LIN {X 0,Y 489.768,Z 496.866,A -85,B 0,C 180,E1 -6554.925,E2 -6554.925} C_VEL
LIN {X 0,Y 489.271,Z 508.598,A -85,B 0,C 180,E1 -6556.29,E2 -6556.29} C_VEL
LIN {X 0,Y 488.822,Z 518.89,A -85,B 0,C 180,E1 -6557.728,E2 -6557.728} C_VEL
LIN {X 0,Y 488.607,Z 527.81,A -85,B 0,C 180,E1 -6559.223,E2 -6559.223} C_VEL
LIN {X 0,Y 488.258,Z 535.963,A -85,B 0,C 180,E1 -6560.89,E2 -6560.89} C_VEL
LIN {X 0,Y 488.146,Z 542.468,A -85,B 0,C 180,E1 -6562.555,E2 -6562.555} C_VEL
LIN {X 0,Y 488.093,Z 547.498,A -85,B 0,C 180,E1 -6564.215,E2 -6564.215} C_VEL
LIN {X 0,Y 488.046,Z 551.175,A -85,B 0,C 180,E1 -6565.871,E2 -6565.871} C_VEL
LIN {X 0,Y 488.011,Z 553.582,A -85,B 0,C 180,E1 -6567.524,E2 -6567.524} C_VEL
LIN {X 0,Y 487.933,Z 554.765,A -85,B 0,C 180,E1 -6569.175,E2 -6569.175} C_VEL
LIN {X 0,Y 487.937,Z 554.732,A -85,B 0,C 180,E1 -6570.825,E2 -6570.825} C_VEL
LIN {X 0,Y 488.021,Z 553.482,A -85,B 0,C 180,E1 -6572.476,E2 -6572.476} C_VEL
LIN {X 0,Y 488.083,Z 551.011,A -85,B 0,C 180,E1 -6574.129,E2 -6574.129} C_VEL
LIN {X 0,Y 488.118,Z 547.258,A -85,B 0,C 180,E1 -6575.785,E2 -6575.785} C_VEL
LIN {X 0,Y 488.183,Z 542.13,A -85,B 0,C 180,E1 -6577.445,E2 -6577.445} C_VEL
LIN {X 0,Y 488.289,Z 535.484,A -85,B 0,C 180,E1 -6579.11,E2 -6579.11} C_VEL
LIN {X 0,Y 488.567,Z 528.339,A -85,B 0,C 180,E1 -6580.569,E2 -6580.569} C_VEL
LIN {X 0,Y 488.758,Z 519.247,A -85,B 0,C 180,E1 -6582.098,E2 -6582.098} C_VEL
LIN {X 0,Y 489.278,Z 507.782,A -85,B 0,C 180,E1 -6583.71,E2 -6583.71} C_VEL
LIN {X 0,Y 489.719,Z 497.109,A -85,B 0,C 180,E1 -6584.971,E2 -6584.971} C_VEL
LIN {X 0,Y 490.258,Z 486.421,A -85,B 0,C 180,E1 -6586.042,E2 -6586.042} C_VEL
LIN {X 0,Y 490.91,Z 472.849,A -85,B 0,C 180,E1 -6587.174,E2 -6587.174} C_VEL
LIN {X 0,Y 491.491,Z 460.708,A -85,B 0,C 180,E1 -6588.013,E2 -6588.013} C_VEL
LIN {X 0,Y 492.097,Z 446.698,A -85,B 0,C 180,E1 -6588.798,E2 -6588.798} C_VEL
LIN {X 0,Y 492.623,Z 432.142,A -85,B 0,C 180,E1 -6589.434,E2 -6589.434} C_VEL
LIN {X 0,Y 493.083,Z 417.146,A -85,B 0,C 180,E1 -6589.914,E2 -6589.914} C_VEL
LIN {X 0,Y 492.97,Z 413.138,A -85,B 0,C 180,E1 -6590.021,E2 -6590.021} C_VEL
LIN {X 0,Y 491.062,Z 401.561,A -85,B 0,C 180,E1 -6590.337,E2 -6590.337} C_VEL
LIN {X 0,Y 489.673,Z 391.28,A -85,B 0,C 180,E1 -6590.556,E2 -6590.556} C_VEL
LIN {X 0,Y 490.143,Z 374.363,A -85,B 0,C 180,E1 -6593.412,E2 -6593.412} C_VEL
LIN {X 0,Y 490.901,Z 356.546,A -85,B 0,C 180,E1 -6596.577,E2 -6596.577} C_VEL
LIN {X 0,Y 491.916,Z 340.726,A -85,B 0,C 180,E1 -6599.609,E2 -6599.609} C_VEL
LIN {X 0,Y 493.222,Z 326.855,A -85,B 0,C 180,E1 -6602.541,E2 -6602.541} C_VEL
LIN {X 0,Y 494.841,Z 316.102,A -85,B 0,C 180,E1 -6605.114,E2 -6605.114} C_VEL
LIN {X 0,Y 494.625,Z 313.33,A -85,B 0,C 180,E1 -6605.914,E2 -6605.914} C_VEL
LIN {X 0,Y 493.242,Z 307.964,A -85,B 0,C 180,E1 -6607.784,E2 -6607.784} C_VEL
LIN {X 0,Y 491.895,Z 302.8,A -85,B 0,C 180,E1 -6610.012,E2 -6610.012} C_VEL
LIN {X 0,Y 490.897,Z 299.006,A -85,B 0,C 180,E1 -6612.29,E2 -6612.29} C_VEL
LIN {X 0,Y 490.311,Z 296.887,A -85,B 0,C 180,E1 -6614.218,E2 -6614.218} C_VEL
LIN {X 0,Y 489.902,Z 295.578,A -85,B 0,C 180,E1 -6616.481,E2 -6616.481} C_VEL
LIN {X 0,Y 489.802,Z 295.249,A -85,B 0,C 180,E1 -6618.697,E2 -6618.697} C_VEL
LIN {X 0,Y 489.783,Z 295.681,A -85,B 0,C 180,E1 -6620.849,E2 -6620.849} C_VEL
LIN {X 0,Y 489.826,Z 296.807,A -85,B 0,C 180,E1 -6623.465,E2 -6623.465} C_VEL
LIN {X 0,Y 489.686,Z 298.58,A -85,B 0,C 180,E1 -6626.349,E2 -6626.349} C_VEL
LIN {X 0,Y 489.42,Z 300.813,A -85,B 0,C 180,E1 -6629.496,E2 -6629.496} C_VEL
LIN {X 0,Y 489.329,Z 302.428,A -85,B 0,C 180,E1 -6631.708,E2 -6631.708} C_VEL
LIN {X 0,Y 489.182,Z 304.804,A -85,B 0,C 180,E1 -6634.839,E2 -6634.839} C_VEL
LIN {X 0,Y 489.027,Z 307.367,A -85,B 0,C 180,E1 -6638.059,E2 -6638.059} C_VEL
LIN {X 0,Y 488.915,Z 309.511,A -85,B 0,C 180,E1 -6640.694,E2 -6640.694} C_VEL
LIN {X 0,Y 488.801,Z 311.695,A -85,B 0,C 180,E1 -6643.288,E2 -6643.288} C_VEL
LIN {X 0,Y 488.772,Z 313.227,A -85,B 0,C 180,E1 -6645.04,E2 -6645.04} C_VEL
LIN {X 0,Y 492.021,Z 323.275,A -85,B 0,C 180,E1 -6645.508,E2 -6645.508} C_VEL
LIN {X 0,Y 491.727,Z 335.772,A -85,B 0,C 180,E1 -6646.044,E2 -6646.044} C_VEL
LIN {X 0,Y 491.293,Z 348.473,A -85,B 0,C 180,E1 -6646.769,E2 -6646.769} C_VEL
LIN {X 0,Y 490.795,Z 359.859,A -85,B 0,C 180,E1 -6647.597,E2 -6647.597} C_VEL
LIN {X 0,Y 490.344,Z 371.117,A -85,B 0,C 180,E1 -6648.634,E2 -6648.634} C_VEL
LIN {X 0,Y 489.981,Z 380.286,A -85,B 0,C 180,E1 -6649.672,E2 -6649.672} C_VEL
LIN {X 0,Y 489.607,Z 387.86,A -85,B 0,C 180,E1 -6650.707,E2 -6650.707} C_VEL
LIN {X 0,Y 489.263,Z 395.396,A -85,B 0,C 180,E1 -6651.97,E2 -6651.97} C_VEL
LIN {X 0,Y 489.024,Z 402.088,A -85,B 0,C 180,E1 -6653.398,E2 -6653.398} C_VEL
LIN {X 0,Y 488.756,Z 406.626,A -85,B 0,C 180,E1 -6654.637,E2 -6654.637} C_VEL
LIN {X 0,Y 488.595,Z 410.068,A -85,B 0,C 180,E1 -6655.876,E2 -6655.876} C_VEL
LIN {X 0,Y 488.644,Z 411.805,A -85,B 0,C 180,E1 -6656.702,E2 -6656.702} C_VEL
LIN {X 0,Y 488.49,Z 413.141,A -85,B 0,C 180,E1 -6657.526,E2 -6657.526} C_VEL
LIN {X 0,Y 488.382,Z 414.052,A -85,B 0,C 180,E1 -6658.351,E2 -6658.351} C_VEL
LIN {X 0,Y 488.402,Z 414.706,A -85,B 0,C 180,E1 -6660,E2 -6660} C_VEL
LIN {X 0,Y 488.403,Z 414.441,A -85,B 0,C 180,E1 -6660.825,E2 -6660.825} C_VEL
LIN {X 0,Y 488.32,Z 412.723,A -85,B 0,C 180,E1 -6662.475,E2 -6662.475} C_VEL
LIN {X 0,Y 488.395,Z 411.27,A -85,B 0,C 180,E1 -6663.3,E2 -6663.3} C_VEL
LIN {X 0,Y 488.539,Z 408.258,A -85,B 0,C 180,E1 -6664.538,E2 -6664.538} C_VEL
LIN {X 0,Y 488.575,Z 404.251,A -85,B 0,C 180,E1 -6665.779,E2 -6665.779} C_VEL
LIN {X 0,Y 488.792,Z 399.728,A -85,B 0,C 180,E1 -6666.879,E2 -6666.879} C_VEL
LIN {X 0,Y 489.007,Z 392.666,A -85,B 0,C 180,E1 -6668.263,E2 -6668.263} C_VEL
LIN {X 0,Y 489.314,Z 384.64,A -85,B 0,C 180,E1 -6669.507,E2 -6669.507} C_VEL
LIN {X 0,Y 489.599,Z 376.5,A -85,B 0,C 180,E1 -6670.546,E2 -6670.546} C_VEL
LIN {X 0,Y 490.05,Z 366.603,A -85,B 0,C 180,E1 -6671.583,E2 -6671.583} C_VEL
LIN {X 0,Y 490.437,Z 355.629,A -85,B 0,C 180,E1 -6672.518,E2 -6672.518} C_VEL
LIN {X 0,Y 490.801,Z 343.259,A -85,B 0,C 180,E1 -6673.35,E2 -6673.35} C_VEL
LIN {X 0,Y 491.123,Z 331.319,A -85,B 0,C 180,E1 -6673.974,E2 -6673.974} C_VEL
LIN {X 0,Y 491.176,Z 320.509,A -85,B 0,C 180,E1 -6674.409,E2 -6674.409} C_VEL
LIN {X 0,Y 488.179,Z 308.882,A -85,B 0,C 180,E1 -6674.859,E2 -6674.859} C_VEL
LIN {X 0,Y 488.179,Z 305.272,A -85,B 0,C 180,E1 -6678.165,E2 -6678.165} C_VEL
LIN {X 0,Y 488.206,Z 302.102,A -85,B 0,C 180,E1 -6681.093,E2 -6681.093} C_VEL
LIN {X 0,Y 488.197,Z 299.235,A -85,B 0,C 180,E1 -6683.771,E2 -6683.771} C_VEL
LIN {X 0,Y 488.232,Z 296.325,A -85,B 0,C 180,E1 -6686.503,E2 -6686.503} C_VEL
LIN {X 0,Y 488.278,Z 293.326,A -85,B 0,C 180,E1 -6689.3,E2 -6689.3} C_VEL
LIN {X 0,Y 488.267,Z 290.293,A -85,B 0,C 180,E1 -6692.179,E2 -6692.179} C_VEL
LIN {X 0,Y 488.605,Z 290.25,A -85,B 0,C 180,E1 -6695.124,E2 -6695.124} C_VEL
LIN {X 0,Y 488.681,Z 290.235,A -85,B 0,C 180,E1 -6698.2,E2 -6698.2} C_VEL
LIN {X 0,Y 488.721,Z 290.231,A -85,B 0,C 180,E1 -6700.345,E2 -6700.345} C_VEL
LIN {X 0,Y 488.687,Z 290.233,A -85,B 0,C 180,E1 -6703.655,E2 -6703.655} C_VEL
LIN {X 0,Y 488.676,Z 290.241,A -85,B 0,C 180,E1 -6706.344,E2 -6706.344} C_VEL
LIN {X 0,Y 488.631,Z 290.247,A -85,B 0,C 180,E1 -6708.576,E2 -6708.576} C_VEL
LIN {X 0,Y 488.638,Z 290.577,A -85,B 0,C 180,E1 -6709.667,E2 -6709.667} C_VEL
LIN {X 0,Y 488.639,Z 294.469,A -85,B 0,C 180,E1 -6712.284,E2 -6712.284} C_VEL
LIN {X 0,Y 488.59,Z 298.405,A -85,B 0,C 180,E1 -6715.075,E2 -6715.075} C_VEL
LIN {X 0,Y 488.542,Z 302.488,A -85,B 0,C 180,E1 -6718.077,E2 -6718.077} C_VEL
LIN {X 0,Y 488.447,Z 305.354,A -85,B 0,C 180,E1 -6720.198,E2 -6720.198} C_VEL
LIN {X 0,Y 487.763,Z 306.347,A -85,B 0,C 180,E1 -6720.877,E2 -6720.877} C_VEL
LIN {X 0,Y 484.894,Z 308.223,A -85,B 0,C 180,E1 -6721.972,E2 -6721.972} C_VEL
LIN {X 0,Y 482.476,Z 309.764,A -85,B 0,C 180,E1 -6722.855,E2 -6722.855} C_VEL
LIN {X 0,Y 481.436,Z 310.86,A -85,B 0,C 180,E1 -6723.538,E2 -6723.538} C_VEL
LIN {X 0,Y 481.351,Z 311.192,A -85,B 0,C 180,E1 -6723.77,E2 -6723.77} C_VEL
LIN {X 0,Y 481.32,Z 315.603,A -85,B 0,C 180,E1 -6726.781,E2 -6726.781} C_VEL
LIN {X 0,Y 481.337,Z 318.973,A -85,B 0,C 180,E1 -6728.946,E2 -6728.946} C_VEL
LIN {X 0,Y 486.935,Z 336.217,A -85,B 0,C 180,E1 -6729.595,E2 -6729.595} C_VEL
LIN {X 0,Y 487.422,Z 339.11,A -85,B 0,C 180,E1 -6729.704,E2 -6729.704} C_VEL
LIN {X 0,Y 487.036,Z 354.063,A -85,B 0,C 180,E1 -6730.234,E2 -6730.234} C_VEL
LIN {X 0,Y 486.428,Z 368.55,A -85,B 0,C 180,E1 -6730.92,E2 -6730.92} C_VEL
LIN {X 0,Y 485.761,Z 382.515,A -85,B 0,C 180,E1 -6731.767,E2 -6731.767} C_VEL
LIN {X 0,Y 485.028,Z 395.249,A -85,B 0,C 180,E1 -6732.72,E2 -6732.72} C_VEL
LIN {X 0,Y 484.313,Z 407.382,A -85,B 0,C 180,E1 -6733.82,E2 -6733.82} C_VEL
LIN {X 0,Y 483.565,Z 418.712,A -85,B 0,C 180,E1 -6735.05,E2 -6735.05} C_VEL
LIN {X 0,Y 482.977,Z 428.555,A -85,B 0,C 180,E1 -6736.322,E2 -6736.322} C_VEL
LIN {X 0,Y 482.399,Z 437.227,A -85,B 0,C 180,E1 -6737.651,E2 -6737.651} C_VEL
LIN {X 0,Y 481.895,Z 446.114,A -85,B 0,C 180,E1 -6739.283,E2 -6739.283} C_VEL
LIN {X 0,Y 481.547,Z 452.691,A -85,B 0,C 180,E1 -6740.761,E2 -6740.761} C_VEL
LIN {X 0,Y 481.289,Z 458.773,A -85,B 0,C 180,E1 -6742.448,E2 -6742.448} C_VEL
LIN {X 0,Y 481.097,Z 463.478,A -85,B 0,C 180,E1 -6744.131,E2 -6744.131} C_VEL
LIN {X 0,Y 480.997,Z 466.926,A -85,B 0,C 180,E1 -6745.81,E2 -6745.81} C_VEL
LIN {X 0,Y 480.935,Z 469.203,A -85,B 0,C 180,E1 -6747.487,E2 -6747.487} C_VEL
LIN {X 0,Y 480.799,Z 470.371,A -85,B 0,C 180,E1 -6749.162,E2 -6749.162} C_VEL
LIN {X 0,Y 480.798,Z 470.387,A -85,B 0,C 180,E1 -6750.837,E2 -6750.837} C_VEL
LIN {X 0,Y 480.935,Z 469.281,A -85,B 0,C 180,E1 -6752.512,E2 -6752.512} C_VEL
LIN {X 0,Y 480.997,Z 467.072,A -85,B 0,C 180,E1 -6754.189,E2 -6754.189} C_VEL
LIN {X 0,Y 481.093,Z 463.7,A -85,B 0,C 180,E1 -6755.869,E2 -6755.869} C_VEL
LIN {X 0,Y 481.287,Z 459.071,A -85,B 0,C 180,E1 -6757.552,E2 -6757.552} C_VEL
LIN {X 0,Y 481.526,Z 453.061,A -85,B 0,C 180,E1 -6759.239,E2 -6759.239} C_VEL
LIN {X 0,Y 481.936,Z 445.488,A -85,B 0,C 180,E1 -6760.928,E2 -6760.928} C_VEL
LIN {X 0,Y 482.375,Z 437.935,A -85,B 0,C 180,E1 -6762.323,E2 -6762.323} C_VEL
LIN {X 0,Y 482.932,Z 429.171,A -85,B 0,C 180,E1 -6763.679,E2 -6763.679} C_VEL
LIN {X 0,Y 483.552,Z 419.434,A -85,B 0,C 180,E1 -6764.95,E2 -6764.95} C_VEL
LIN {X 0,Y 484.243,Z 408.371,A -85,B 0,C 180,E1 -6766.17,E2 -6766.17} C_VEL
LIN {X 0,Y 485.004,Z 396.286,A -85,B 0,C 180,E1 -6767.281,E2 -6767.281} C_VEL
LIN {X 0,Y 485.703,Z 383.774,A -85,B 0,C 180,E1 -6768.234,E2 -6768.234} C_VEL
LIN {X 0,Y 486.312,Z 370.13,A -85,B 0,C 180,E1 -6769.085,E2 -6769.085} C_VEL
LIN {X 0,Y 486.971,Z 355.986,A -85,B 0,C 180,E1 -6769.774,E2 -6769.774} C_VEL
LIN {X 0,Y 487.378,Z 341.683,A -85,B 0,C 180,E1 -6770.306,E2 -6770.306} C_VEL
LIN {X 0,Y 487.231,Z 337.436,A -85,B 0,C 180,E1 -6770.449,E2 -6770.449} C_VEL
LIN {X 0,Y 483.022,Z 324.071,A -85,B 0,C 180,E1 -6770.962,E2 -6770.962} C_VEL
LIN {X 0,Y 481.339,Z 318.996,A -85,B 0,C 180,E1 -6771.14,E2 -6771.14} C_VEL
LIN {X 0,Y 481.312,Z 314.379,A -85,B 0,C 180,E1 -6774.132,E2 -6774.132} C_VEL
LIN {X 0,Y 481.401,Z 310.161,A -85,B 0,C 180,E1 -6777.058,E2 -6777.058} C_VEL
LIN {X 0,Y 481.418,Z 306.456,A -85,B 0,C 180,E1 -6779.759,E2 -6779.759} C_VEL
LIN {X 0,Y 481.49,Z 302.545,A -85,B 0,C 180,E1 -6782.688,E2 -6782.688} C_VEL
LIN {X 0,Y 481.548,Z 298.434,A -85,B 0,C 180,E1 -6785.717,E2 -6785.717} C_VEL
LIN {X 0,Y 481.643,Z 293.949,A -85,B 0,C 180,E1 -6788.862,E2 -6788.862} C_VEL
LIN {X 0,Y 481.548,Z 291.136,A -85,B 0,C 180,E1 -6790.806,E2 -6790.806} C_VEL
LIN {X 0,Y 481.622,Z 291.12,A -85,B 0,C 180,E1 -6793.302,E2 -6793.302} C_VEL
LIN {X 0,Y 481.659,Z 291.116,A -85,B 0,C 180,E1 -6795.641,E2 -6795.641} C_VEL
LIN {X 0,Y 481.657,Z 291.114,A -85,B 0,C 180,E1 -6798.958,E2 -6798.958} C_VEL
LIN {X 0,Y 481.652,Z 291.117,A -85,B 0,C 180,E1 -6801.993,E2 -6801.993} C_VEL
LIN {X 0,Y 481.691,Z 291.111,A -85,B 0,C 180,E1 -6805.318,E2 -6805.318} C_VEL
LIN {X 0,Y 481.644,Z 291.116,A -85,B 0,C 180,E1 -6808.311,E2 -6808.311} C_VEL
LIN {X 0,Y 481.657,Z 291.111,A -85,B 0,C 180,E1 -6811.216,E2 -6811.216} C_VEL
LIN {X 0,Y 481.646,Z 291.11,A -85,B 0,C 180,E1 -6814.04,E2 -6814.04} C_VEL
LIN {X 0,Y 481.675,Z 291.113,A -85,B 0,C 180,E1 -6816.812,E2 -6816.812} C_VEL
LIN {X 0,Y 481.695,Z 291.104,A -85,B 0,C 180,E1 -6819.503,E2 -6819.503} C_VEL
LIN {X 0,Y 481.682,Z 291.105,A -85,B 0,C 180,E1 -6822.157,E2 -6822.157} C_VEL
LIN {X 0,Y 481.745,Z 291.099,A -85,B 0,C 180,E1 -6824.776,E2 -6824.776} C_VEL
LIN {X 0,Y 481.752,Z 291.095,A -85,B 0,C 180,E1 -6828.215,E2 -6828.215} C_VEL
LIN {X 0,Y 481.73,Z 291.105,A -85,B 0,C 180,E1 -6831.611,E2 -6831.611} C_VEL
LIN {X 0,Y 481.786,Z 291.089,A -85,B 0,C 180,E1 -6834.139,E2 -6834.139} C_VEL
LIN {X 0,Y 481.926,Z 291.077,A -85,B 0,C 180,E1 -6837.492,E2 -6837.492} C_VEL
LIN {X 0,Y 481.942,Z 291.069,A -85,B 0,C 180,E1 -6840,E2 -6840} C_VEL
LIN {X 0,Y 481.918,Z 291.079,A -85,B 0,C 180,E1 -6842.507,E2 -6842.507} C_VEL
LIN {X 0,Y 481.785,Z 291.09,A -85,B 0,C 180,E1 -6845.861,E2 -6845.861} C_VEL
LIN {X 0,Y 481.742,Z 291.104,A -85,B 0,C 180,E1 -6848.389,E2 -6848.389} C_VEL
LIN {X 0,Y 481.751,Z 291.094,A -85,B 0,C 180,E1 -6851.785,E2 -6851.785} C_VEL
LIN {X 0,Y 481.738,Z 291.101,A -85,B 0,C 180,E1 -6855.224,E2 -6855.224} C_VEL
LIN {X 0,Y 481.709,Z 291.109,A -85,B 0,C 180,E1 -6858.722,E2 -6858.722} C_VEL
LIN {X 0,Y 481.646,Z 291.108,A -85,B 0,C 180,E1 -6861.395,E2 -6861.395} C_VEL
LIN {X 0,Y 481.648,Z 291.113,A -85,B 0,C 180,E1 -6864.115,E2 -6864.115} C_VEL
LIN {X 0,Y 481.675,Z 291.108,A -85,B 0,C 180,E1 -6867.122,E2 -6867.122} C_VEL
LIN {X 0,Y 481.673,Z 291.11,A -85,B 0,C 180,E1 -6869.741,E2 -6869.741} C_VEL
LIN {X 0,Y 481.672,Z 291.109,A -85,B 0,C 180,E1 -6872.674,E2 -6872.674} C_VEL
LIN {X 0,Y 481.66,Z 291.115,A -85,B 0,C 180,E1 -6875.204,E2 -6875.204} C_VEL
LIN {X 0,Y 481.666,Z 291.113,A -85,B 0,C 180,E1 -6878.859,E2 -6878.859} C_VEL
LIN {X 0,Y 481.652,Z 291.112,A -85,B 0,C 180,E1 -6881.913,E2 -6881.913} C_VEL
LIN {X 0,Y 481.654,Z 291.109,A -85,B 0,C 180,E1 -6884.458,E2 -6884.458} C_VEL
LIN {X 0,Y 481.628,Z 291.112,A -85,B 0,C 180,E1 -6887.837,E2 -6887.837} C_VEL
LIN {X 0,Y 481.646,Z 291.215,A -85,B 0,C 180,E1 -6888.591,E2 -6888.591} C_VEL
LIN {X 0,Y 484.909,Z 303.856,A -85,B 0,C 180,E1 -6891.801,E2 -6891.801} C_VEL
LIN {X 0,Y 487.48,Z 314.226,A -85,B 0,C 180,E1 -6894.278,E2 -6894.278} C_VEL
LIN {X 0,Y 487.662,Z 316.627,A -85,B 0,C 180,E1 -6894.798,E2 -6894.798} C_VEL
LIN {X 0,Y 486.351,Z 332.215,A -85,B 0,C 180,E1 -6897.924,E2 -6897.924} C_VEL
LIN {X 0,Y 485.178,Z 347.976,A -85,B 0,C 180,E1 -6900.971,E2 -6900.971} C_VEL
LIN {X 0,Y 484.134,Z 365.065,A -85,B 0,C 180,E1 -6904.162,E2 -6904.162} C_VEL
LIN {X 0,Y 483.249,Z 382.552,A -85,B 0,C 180,E1 -6907.332,E2 -6907.332} C_VEL
LIN {X 0,Y 482.896,Z 392.937,A -85,B 0,C 180,E1 -6909.176,E2 -6909.176} C_VEL
LIN {X 0,Y 485.472,Z 409.983,A -85,B 0,C 180,E1 -6909.592,E2 -6909.592} C_VEL
LIN {X 0,Y 486.389,Z 416.005,A -85,B 0,C 180,E1 -6909.781,E2 -6909.781} C_VEL
LIN {X 0,Y 485.948,Z 429.67,A -85,B 0,C 180,E1 -6910.213,E2 -6910.213} C_VEL
LIN {X 0,Y 485.389,Z 443.979,A -85,B 0,C 180,E1 -6910.823,E2 -6910.823} C_VEL
LIN {X 0,Y 484.694,Z 458.387,A -85,B 0,C 180,E1 -6911.617,E2 -6911.617} C_VEL
LIN {X 0,Y 484.002,Z 472.236,A -85,B 0,C 180,E1 -6912.573,E2 -6912.573} C_VEL
LIN {X 0,Y 483.374,Z 485.225,A -85,B 0,C 180,E1 -6913.659,E2 -6913.659} C_VEL
LIN {X 0,Y 482.742,Z 496.737,A -85,B 0,C 180,E1 -6914.808,E2 -6914.808} C_VEL
LIN {X 0,Y 482.237,Z 507.517,A -85,B 0,C 180,E1 -6916.086,E2 -6916.086} C_VEL
LIN {X 0,Y 481.751,Z 518.228,A -85,B 0,C 180,E1 -6917.604,E2 -6917.604} C_VEL
LIN {X 0,Y 481.501,Z 526.782,A -85,B 0,C 180,E1 -6919.062,E2 -6919.062} C_VEL
LIN {X 0,Y 481.199,Z 534.958,A -85,B 0,C 180,E1 -6920.755,E2 -6920.755} C_VEL
LIN {X 0,Y 481.078,Z 541.48,A -85,B 0,C 180,E1 -6922.445,E2 -6922.445} C_VEL
LIN {X 0,Y 481.041,Z 546.52,A -85,B 0,C 180,E1 -6924.13,E2 -6924.13} C_VEL
LIN {X 0,Y 480.989,Z 550.199,A -85,B 0,C 180,E1 -6925.811,E2 -6925.811} C_VEL
LIN {X 0,Y 480.97,Z 552.608,A -85,B 0,C 180,E1 -6927.488,E2 -6927.488} C_VEL
LIN {X 0,Y 480.9,Z 553.788,A -85,B 0,C 180,E1 -6929.163,E2 -6929.163} C_VEL
LIN {X 0,Y 480.906,Z 553.741,A -85,B 0,C 180,E1 -6930.838,E2 -6930.838} C_VEL
LIN {X 0,Y 480.985,Z 552.471,A -85,B 0,C 180,E1 -6932.513,E2 -6932.513} C_VEL
LIN {X 0,Y 481.059,Z 549.976,A -85,B 0,C 180,E1 -6934.189,E2 -6934.189} C_VEL
LIN {X 0,Y 481.072,Z 546.188,A -85,B 0,C 180,E1 -6935.87,E2 -6935.87} C_VEL
LIN {X 0,Y 481.129,Z 541.02,A -85,B 0,C 180,E1 -6937.555,E2 -6937.555} C_VEL
LIN {X 0,Y 481.224,Z 534.358,A -85,B 0,C 180,E1 -6939.245,E2 -6939.245} C_VEL
LIN {X 0,Y 481.518,Z 526.248,A -85,B 0,C 180,E1 -6940.938,E2 -6940.938} C_VEL
LIN {X 0,Y 481.778,Z 517.266,A -85,B 0,C 180,E1 -6942.475,E2 -6942.475} C_VEL
LIN {X 0,Y 482.268,Z 507.162,A -85,B 0,C 180,E1 -6943.913,E2 -6943.913} C_VEL
LIN {X 0,Y 482.757,Z 496.491,A -85,B 0,C 180,E1 -6945.192,E2 -6945.192} C_VEL
LIN {X 0,Y 483.417,Z 484.904,A -85,B 0,C 180,E1 -6946.359,E2 -6946.359} C_VEL
LIN {X 0,Y 484.035,Z 472.246,A -85,B 0,C 180,E1 -6947.426,E2 -6947.426} C_VEL
LIN {X 0,Y 484.667,Z 460.108,A -85,B 0,C 180,E1 -6948.275,E2 -6948.275} C_VEL
LIN {X 0,Y 485.322,Z 446.106,A -85,B 0,C 180,E1 -6949.071,E2 -6949.071} C_VEL
LIN {X 0,Y 485.848,Z 432.317,A -85,B 0,C 180,E1 -6949.685,E2 -6949.685} C_VEL
LIN {X 0,Y 486.349,Z 417.616,A -85,B 0,C 180,E1 -6950.171,E2 -6950.171} C_VEL
LIN {X 0,Y 486.297,Z 414.548,A -85,B 0,C 180,E1 -6950.26,E2 -6950.26} C_VEL
LIN {X 0,Y 484.394,Z 402.571,A -85,B 0,C 180,E1 -6950.602,E2 -6950.602} C_VEL
LIN {X 0,Y 482.66,Z 390.05,A -85,B 0,C 180,E1 -6950.901,E2 -6950.901} C_VEL
LIN {X 0,Y 483.195,Z 373.568,A -85,B 0,C 180,E1 -6953.761,E2 -6953.761} C_VEL
LIN {X 0,Y 483.978,Z 357.186,A -85,B 0,C 180,E1 -6956.754,E2 -6956.754} C_VEL
LIN {X 0,Y 484.979,Z 342.672,A -85,B 0,C 180,E1 -6959.602,E2 -6959.602} C_VEL
LIN {X 0,Y 486.225,Z 329.979,A -85,B 0,C 180,E1 -6962.331,E2 -6962.331} C_VEL
LIN {X 0,Y 487.828,Z 319.704,A -85,B 0,C 180,E1 -6964.797,E2 -6964.797} C_VEL
LIN {X 0,Y 488.123,Z 316.525,A -85,B 0,C 180,E1 -6965.666,E2 -6965.666} C_VEL
LIN {X 0,Y 486.836,Z 311.322,A -85,B 0,C 180,E1 -6967.441,E2 -6967.441} C_VEL
LIN {X 0,Y 485.515,Z 306.272,A -85,B 0,C 180,E1 -6969.563,E2 -6969.563} C_VEL
LIN {X 0,Y 484.441,Z 302.12,A -85,B 0,C 180,E1 -6971.863,E2 -6971.863} C_VEL
LIN {X 0,Y 483.644,Z 299.298,A -85,B 0,C 180,E1 -6974.228,E2 -6974.228} C_VEL
LIN {X 0,Y 483.154,Z 297.722,A -85,B 0,C 180,E1 -6976.869,E2 -6976.869} C_VEL
LIN {X 0,Y 483.012,Z 297.409,A -85,B 0,C 180,E1 -6979.167,E2 -6979.167} C_VEL
LIN {X 0,Y 482.949,Z 298.133,A -85,B 0,C 180,E1 -6982.324,E2 -6982.324} C_VEL
LIN {X 0,Y 482.881,Z 299.204,A -85,B 0,C 180,E1 -6984.592,E2 -6984.592} C_VEL
LIN {X 0,Y 482.768,Z 300.278,A -85,B 0,C 180,E1 -6986.414,E2 -6986.414} C_VEL
LIN {X 0,Y 482.499,Z 302.207,A -85,B 0,C 180,E1 -6989.349,E2 -6989.349} C_VEL
LIN {X 0,Y 482.346,Z 304.273,A -85,B 0,C 180,E1 -6992.209,E2 -6992.209} C_VEL
LIN {X 0,Y 482.214,Z 306.359,A -85,B 0,C 180,E1 -6994.998,E2 -6994.998} C_VEL
LIN {X 0,Y 482.075,Z 308.443,A -85,B 0,C 180,E1 -6997.726,E2 -6997.726} C_VEL
LIN {X 0,Y 481.967,Z 310.587,A -85,B 0,C 180,E1 -7000.404,E2 -7000.404} C_VEL
LIN {X 0,Y 481.828,Z 312.792,A -85,B 0,C 180,E1 -7003.039,E2 -7003.039} C_VEL
LIN {X 0,Y 481.786,Z 314.259,A -85,B 0,C 180,E1 -7004.738,E2 -7004.738} C_VEL
LIN {X 0,Y 485.354,Z 324.672,A -85,B 0,C 180,E1 -7005.268,E2 -7005.268} C_VEL
LIN {X 0,Y 484.99,Z 337.668,A -85,B 0,C 180,E1 -7005.846,E2 -7005.846} C_VEL
LIN {X 0,Y 484.542,Z 350.118,A -85,B 0,C 180,E1 -7006.581,E2 -7006.581} C_VEL
LIN {X 0,Y 484.008,Z 361.343,A -85,B 0,C 180,E1 -7007.42,E2 -7007.42} C_VEL
LIN {X 0,Y 483.503,Z 372.495,A -85,B 0,C 180,E1 -7008.471,E2 -7008.471} C_VEL
LIN {X 0,Y 483.125,Z 381.556,A -85,B 0,C 180,E1 -7009.523,E2 -7009.523} C_VEL
LIN {X 0,Y 482.593,Z 390.404,A -85,B 0,C 180,E1 -7010.782,E2 -7010.782} C_VEL
LIN {X 0,Y 482.277,Z 397.716,A -85,B 0,C 180,E1 -7012.085,E2 -7012.085} C_VEL
LIN {X 0,Y 482.068,Z 403.22,A -85,B 0,C 180,E1 -7013.302,E2 -7013.302} C_VEL
LIN {X 0,Y 481.786,Z 407.742,A -85,B 0,C 180,E1 -7014.559,E2 -7014.559} C_VEL
LIN {X 0,Y 481.601,Z 411.173,A -85,B 0,C 180,E1 -7015.816,E2 -7015.816} C_VEL
LIN {X 0,Y 481.644,Z 412.899,A -85,B 0,C 180,E1 -7016.654,E2 -7016.654} C_VEL
LIN {X 0,Y 481.485,Z 414.224,A -85,B 0,C 180,E1 -7017.49,E2 -7017.49} C_VEL
LIN {X 0,Y 481.407,Z 415.624,A -85,B 0,C 180,E1 -7019.164,E2 -7019.164} C_VEL
LIN {X 0,Y 481.39,Z 415.747,A -85,B 0,C 180,E1 -7020,E2 -7020} C_VEL
LIN {X 0,Y 481.393,Z 415.466,A -85,B 0,C 180,E1 -7020.837,E2 -7020.837} C_VEL
LIN {X 0,Y 481.298,Z 413.721,A -85,B 0,C 180,E1 -7022.511,E2 -7022.511} C_VEL
LIN {X 0,Y 481.373,Z 412.241,A -85,B 0,C 180,E1 -7023.348,E2 -7023.348} C_VEL
LIN {X 0,Y 481.53,Z 409.199,A -85,B 0,C 180,E1 -7024.604,E2 -7024.604} C_VEL
LIN {X 0,Y 481.579,Z 405.157,A -85,B 0,C 180,E1 -7025.863,E2 -7025.863} C_VEL
LIN {X 0,Y 481.86,Z 398.913,A -85,B 0,C 180,E1 -7027.345,E2 -7027.345} C_VEL
LIN {X 0,Y 482.13,Z 392.238,A -85,B 0,C 180,E1 -7028.593,E2 -7028.593} C_VEL
LIN {X 0,Y 482.389,Z 383.925,A -85,B 0,C 180,E1 -7029.857,E2 -7029.857} C_VEL
LIN {X 0,Y 482.773,Z 375.444,A -85,B 0,C 180,E1 -7030.909,E2 -7030.909} C_VEL
LIN {X 0,Y 483.193,Z 365.07,A -85,B 0,C 180,E1 -7031.962,E2 -7031.962} C_VEL
LIN {X 0,Y 483.609,Z 353.726,A -85,B 0,C 180,E1 -7032.893,E2 -7032.893} C_VEL
LIN {X 0,Y 483.998,Z 342.2,A -85,B 0,C 180,E1 -7033.648,E2 -7033.648} C_VEL
LIN {X 0,Y 484.351,Z 329.624,A -85,B 0,C 180,E1 -7034.281,E2 -7034.281} C_VEL
LIN {X 0,Y 484.316,Z 321.621,A -85,B 0,C 180,E1 -7034.604,E2 -7034.604} C_VEL
LIN {X 0,Y 481.14,Z 309.388,A -85,B 0,C 180,E1 -7035.108,E2 -7035.108} C_VEL
LIN {X 0,Y 481.135,Z 305.898,A -85,B 0,C 180,E1 -7038.292,E2 -7038.292} C_VEL
LIN {X 0,Y 481.143,Z 302.508,A -85,B 0,C 180,E1 -7041.418,E2 -7041.418} C_VEL
LIN {X 0,Y 481.162,Z 299.591,A -85,B 0,C 180,E1 -7044.141,E2 -7044.141} C_VEL
LIN {X 0,Y 481.173,Z 296.539,A -85,B 0,C 180,E1 -7047.005,E2 -7047.005} C_VEL
LIN {X 0,Y 481.224,Z 293.574,A -85,B 0,C 180,E1 -7049.772,E2 -7049.772} C_VEL
LIN {X 0,Y 481.234,Z 291.169,A -85,B 0,C 180,E1 -7052.108,E2 -7052.108} C_VEL
LIN {X 0,Y 481.559,Z 291.128,A -85,B 0,C 180,E1 -7055.186,E2 -7055.186} C_VEL
LIN {X 0,Y 481.653,Z 291.111,A -85,B 0,C 180,E1 -7058.006,E2 -7058.006} C_VEL
LIN {X 0,Y 481.659,Z 291.111,A -85,B 0,C 180,E1 -7061.042,E2 -7061.042} C_VEL
LIN {X 0,Y 481.657,Z 291.113,A -85,B 0,C 180,E1 -7064.458,E2 -7064.458} C_VEL
LIN {X 0,Y 481.618,Z 291.118,A -85,B 0,C 180,E1 -7066.855,E2 -7066.855} C_VEL
LIN {X 0,Y 481.552,Z 291.148,A -85,B 0,C 180,E1 -7069.369,E2 -7069.369} C_VEL
LIN {X 0,Y 481.619,Z 295.035,A -85,B 0,C 180,E1 -7071.998,E2 -7071.998} C_VEL
LIN {X 0,Y 481.561,Z 299.679,A -85,B 0,C 180,E1 -7075.307,E2 -7075.307} C_VEL
LIN {X 0,Y 481.475,Z 303.731,A -85,B 0,C 180,E1 -7078.299,E2 -7078.299} C_VEL
LIN {X 0,Y 481.408,Z 307.643,A -85,B 0,C 180,E1 -7081.199,E2 -7081.199} C_VEL
LIN {X 0,Y 481.351,Z 311.192,A -85,B 0,C 180,E1 -7083.77,E2 -7083.77} C_VEL
LIN {X 0,Y 480.681,Z 312.262,A -85,B 0,C 180,E1 -7084.456,E2 -7084.456} C_VEL
LIN {X 0,Y 477.821,Z 314.277,A -85,B 0,C 180,E1 -7085.564,E2 -7085.564} C_VEL
LIN {X 0,Y 475.399,Z 315.968,A -85,B 0,C 180,E1 -7086.456,E2 -7086.456} C_VEL
LIN {X 0,Y 474.355,Z 317.173,A -85,B 0,C 180,E1 -7087.147,E2 -7087.147} C_VEL
LIN {X 0,Y 474.267,Z 317.544,A -85,B 0,C 180,E1 -7087.381,E2 -7087.381} C_VEL
LIN {X 0,Y 474.313,Z 319.528,A -85,B 0,C 180,E1 -7088.627,E2 -7088.627} C_VEL
LIN {X 0,Y 479.666,Z 335.669,A -85,B 0,C 180,E1 -7089.241,E2 -7089.241} C_VEL
LIN {X 0,Y 480.784,Z 340.036,A -85,B 0,C 180,E1 -7089.423,E2 -7089.423} C_VEL
LIN {X 0,Y 480.385,Z 355.019,A -85,B 0,C 180,E1 -7089.965,E2 -7089.965} C_VEL
LIN {X 0,Y 479.739,Z 369.145,A -85,B 0,C 180,E1 -7090.643,E2 -7090.643} C_VEL
LIN {X 0,Y 479.071,Z 383.112,A -85,B 0,C 180,E1 -7091.504,E2 -7091.504} C_VEL
LIN {X 0,Y 478.294,Z 395.85,A -85,B 0,C 180,E1 -7092.469,E2 -7092.469} C_VEL
LIN {X 0,Y 477.521,Z 408.05,A -85,B 0,C 180,E1 -7093.59,E2 -7093.59} C_VEL
LIN {X 0,Y 476.732,Z 419.318,A -85,B 0,C 180,E1 -7094.831,E2 -7094.831} C_VEL
LIN {X 0,Y 476.106,Z 429.161,A -85,B 0,C 180,E1 -7096.121,E2 -7096.121} C_VEL
LIN {X 0,Y 475.468,Z 438.068,A -85,B 0,C 180,E1 -7097.507,E2 -7097.507} C_VEL
LIN {X 0,Y 474.933,Z 446.723,A -85,B 0,C 180,E1 -7099.124,E2 -7099.124} C_VEL
LIN {X 0,Y 474.563,Z 453.299,A -85,B 0,C 180,E1 -7100.624,E2 -7100.624} C_VEL
LIN {X 0,Y 474.258,Z 459.383,A -85,B 0,C 180,E1 -7102.335,E2 -7102.335} C_VEL
LIN {X 0,Y 474.05,Z 464.087,A -85,B 0,C 180,E1 -7104.043,E2 -7104.043} C_VEL
LIN {X 0,Y 473.946,Z 467.535,A -85,B 0,C 180,E1 -7105.748,E2 -7105.748} C_VEL
LIN {X 0,Y 473.878,Z 469.811,A -85,B 0,C 180,E1 -7107.45,E2 -7107.45} C_VEL
LIN {X 0,Y 473.726,Z 470.98,A -85,B 0,C 180,E1 -7109.15,E2 -7109.15} C_VEL
LIN {X 0,Y 473.726,Z 470.996,A -85,B 0,C 180,E1 -7110.85,E2 -7110.85} C_VEL
LIN {X 0,Y 473.878,Z 469.888,A -85,B 0,C 180,E1 -7112.55,E2 -7112.55} C_VEL
LIN {X 0,Y 473.946,Z 467.678,A -85,B 0,C 180,E1 -7114.252,E2 -7114.252} C_VEL
LIN {X 0,Y 474.046,Z 464.306,A -85,B 0,C 180,E1 -7115.957,E2 -7115.957} C_VEL
LIN {X 0,Y 474.253,Z 459.676,A -85,B 0,C 180,E1 -7117.664,E2 -7117.664} C_VEL
LIN {X 0,Y 474.543,Z 453.663,A -85,B 0,C 180,E1 -7119.376,E2 -7119.376} C_VEL
LIN {X 0,Y 474.98,Z 446.09,A -85,B 0,C 180,E1 -7121.09,E2 -7121.09} C_VEL
LIN {X 0,Y 475.425,Z 438.751,A -85,B 0,C 180,E1 -7122.47,E2 -7122.47} C_VEL
LIN {X 0,Y 476.035,Z 429.771,A -85,B 0,C 180,E1 -7123.881,E2 -7123.881} C_VEL
LIN {X 0,Y 476.715,Z 420.031,A -85,B 0,C 180,E1 -7125.17,E2 -7125.17} C_VEL
LIN {X 0,Y 477.445,Z 409.04,A -85,B 0,C 180,E1 -7126.398,E2 -7126.398} C_VEL
LIN {X 0,Y 478.255,Z 396.876,A -85,B 0,C 180,E1 -7127.532,E2 -7127.532} C_VEL
LIN {X 0,Y 479.006,Z 384.357,A -85,B 0,C 180,E1 -7128.499,E2 -7128.499} C_VEL
LIN {X 0,Y 479.645,Z 370.706,A -85,B 0,C 180,E1 -7129.36,E2 -7129.36} C_VEL
LIN {X 0,Y 480.323,Z 355.736,A -85,B 0,C 180,E1 -7130.097,E2 -7130.097} C_VEL
LIN {X 0,Y 480.769,Z 341.195,A -85,B 0,C 180,E1 -7130.631,E2 -7130.631} C_VEL
LIN {X 0,Y 480.497,Z 338.377,A -85,B 0,C 180,E1 -7130.736,E2 -7130.736} C_VEL
LIN {X 0,Y 476.491,Z 326.04,A -85,B 0,C 180,E1 -7131.232,E2 -7131.232} C_VEL
LIN {X 0,Y 474.302,Z 319.532,A -85,B 0,C 180,E1 -7131.467,E2 -7131.467} C_VEL
LIN {X 0,Y 474.305,Z 314.816,A -85,B 0,C 180,E1 -7134.512,E2 -7134.512} C_VEL
LIN {X 0,Y 474.384,Z 310.749,A -85,B 0,C 180,E1 -7137.34,E2 -7137.34} C_VEL
LIN {X 0,Y 474.386,Z 306.763,A -85,B 0,C 180,E1 -7140.245,E2 -7140.245} C_VEL
LIN {X 0,Y 474.478,Z 302.761,A -85,B 0,C 180,E1 -7143.233,E2 -7143.233} C_VEL
LIN {X 0,Y 474.536,Z 298.548,A -85,B 0,C 180,E1 -7146.328,E2 -7146.328} C_VEL
LIN {X 0,Y 474.594,Z 295.524,A -85,B 0,C 180,E1 -7148.459,E2 -7148.459} C_VEL
LIN {X 0,Y 474.537,Z 292.01,A -85,B 0,C 180,E1 -7150.946,E2 -7150.946} C_VEL
LIN {X 0,Y 474.605,Z 291.994,A -85,B 0,C 180,E1 -7154.105,E2 -7154.105} C_VEL
LIN {X 0,Y 474.615,Z 291.994,A -85,B 0,C 180,E1 -7157.066,E2 -7157.066} C_VEL
LIN {X 0,Y 474.617,Z 291.989,A -85,B 0,C 180,E1 -7159.342,E2 -7159.342} C_VEL
LIN {X 0,Y 474.589,Z 291.992,A -85,B 0,C 180,E1 -7162.616,E2 -7162.616} C_VEL
LIN {X 0,Y 474.633,Z 291.986,A -85,B 0,C 180,E1 -7165.759,E2 -7165.759} C_VEL
LIN {X 0,Y 474.597,Z 291.992,A -85,B 0,C 180,E1 -7168.782,E2 -7168.782} C_VEL
LIN {X 0,Y 474.602,Z 291.993,A -85,B 0,C 180,E1 -7171.715,E2 -7171.715} C_VEL
LIN {X 0,Y 474.628,Z 291.983,A -85,B 0,C 180,E1 -7174.589,E2 -7174.589} C_VEL
LIN {X 0,Y 474.6,Z 291.987,A -85,B 0,C 180,E1 -7177.355,E2 -7177.355} C_VEL
LIN {X 0,Y 474.652,Z 291.986,A -85,B 0,C 180,E1 -7180.089,E2 -7180.089} C_VEL
LIN {X 0,Y 474.627,Z 291.98,A -85,B 0,C 180,E1 -7182.773,E2 -7182.773} C_VEL
LIN {X 0,Y 474.653,Z 291.988,A -85,B 0,C 180,E1 -7185.421,E2 -7185.421} C_VEL
LIN {X 0,Y 474.705,Z 291.972,A -85,B 0,C 180,E1 -7188.038,E2 -7188.038} C_VEL
LIN {X 0,Y 474.704,Z 291.979,A -85,B 0,C 180,E1 -7191.486,E2 -7191.486} C_VEL
LIN {X 0,Y 474.747,Z 291.965,A -85,B 0,C 180,E1 -7194.052,E2 -7194.052} C_VEL
LIN {X 0,Y 474.892,Z 291.953,A -85,B 0,C 180,E1 -7197.455,E2 -7197.455} C_VEL
LIN {X 0,Y 474.913,Z 291.944,A -85,B 0,C 180,E1 -7200,E2 -7200} C_VEL
LIN {X 0,Y 474.883,Z 291.955,A -85,B 0,C 180,E1 -7202.545,E2 -7202.545} C_VEL
LIN {X 0,Y 474.75,Z 291.966,A -85,B 0,C 180,E1 -7205.948,E2 -7205.948} C_VEL
LIN {X 0,Y 474.713,Z 291.981,A -85,B 0,C 180,E1 -7208.514,E2 -7208.514} C_VEL
LIN {X 0,Y 474.705,Z 291.974,A -85,B 0,C 180,E1 -7211.962,E2 -7211.962} C_VEL
LIN {X 0,Y 474.679,Z 291.974,A -85,B 0,C 180,E1 -7215.767,E2 -7215.767} C_VEL
LIN {X 0,Y 474.663,Z 291.984,A -85,B 0,C 180,E1 -7219.01,E2 -7219.01} C_VEL
LIN {X 0,Y 474.588,Z 291.987,A -85,B 0,C 180,E1 -7221.729,E2 -7221.729} C_VEL
LIN {X 0,Y 474.626,Z 291.988,A -85,B 0,C 180,E1 -7224.495,E2 -7224.495} C_VEL
LIN {X 0,Y 474.636,Z 291.985,A -85,B 0,C 180,E1 -7227.324,E2 -7227.324} C_VEL
LIN {X 0,Y 474.603,Z 291.995,A -85,B 0,C 180,E1 -7230.23,E2 -7230.23} C_VEL
LIN {X 0,Y 474.642,Z 291.987,A -85,B 0,C 180,E1 -7233.22,E2 -7233.22} C_VEL
LIN {X 0,Y 474.583,Z 291.993,A -85,B 0,C 180,E1 -7236.324,E2 -7236.324} C_VEL
LIN {X 0,Y 474.615,Z 291.99,A -85,B 0,C 180,E1 -7239.646,E2 -7239.646} C_VEL
LIN {X 0,Y 474.624,Z 291.986,A -85,B 0,C 180,E1 -7242.237,E2 -7242.237} C_VEL
LIN {X 0,Y 474.615,Z 291.986,A -85,B 0,C 180,E1 -7245.298,E2 -7245.298} C_VEL
LIN {X 0,Y 474.624,Z 292.086,A -85,B 0,C 180,E1 -7248.105,E2 -7248.105} C_VEL
LIN {X 0,Y 477.33,Z 302.647,A -85,B 0,C 180,E1 -7250.875,E2 -7250.875} C_VEL
LIN {X 0,Y 480.295,Z 314.533,A -85,B 0,C 180,E1 -7253.787,E2 -7253.787} C_VEL
LIN {X 0,Y 480.893,Z 318.339,A -85,B 0,C 180,E1 -7254.661,E2 -7254.661} C_VEL
LIN {X 0,Y 479.451,Z 334.239,A -85,B 0,C 180,E1 -7257.902,E2 -7257.902} C_VEL
LIN {X 0,Y 478.217,Z 349.953,A -85,B 0,C 180,E1 -7260.989,E2 -7260.989} C_VEL
LIN {X 0,Y 477.182,Z 366.044,A -85,B 0,C 180,E1 -7264.056,E2 -7264.056} C_VEL
LIN {X 0,Y 476.205,Z 384.364,A -85,B 0,C 180,E1 -7267.436,E2 -7267.436} C_VEL
LIN {X 0,Y 475.88,Z 392.154,A -85,B 0,C 180,E1 -7268.846,E2 -7268.846} C_VEL
LIN {X 0,Y 478.821,Z 411.414,A -85,B 0,C 180,E1 -7269.347,E2 -7269.347} C_VEL
LIN {X 0,Y 479.675,Z 417.083,A -85,B 0,C 180,E1 -7269.536,E2 -7269.536} C_VEL
LIN {X 0,Y 479.162,Z 430.777,A -85,B 0,C 180,E1 -7269.987,E2 -7269.987} C_VEL
LIN {X 0,Y 478.535,Z 445.519,A -85,B 0,C 180,E1 -7270.649,E2 -7270.649} C_VEL
LIN {X 0,Y 477.807,Z 459.5,A -85,B 0,C 180,E1 -7271.453,E2 -7271.453} C_VEL
LIN {X 0,Y 477.061,Z 473.038,A -85,B 0,C 180,E1 -7272.422,E2 -7272.422} C_VEL
LIN {X 0,Y 476.368,Z 486.339,A -85,B 0,C 180,E1 -7273.59,E2 -7273.59} C_VEL
LIN {X 0,Y 475.686,Z 497.817,A -85,B 0,C 180,E1 -7274.797,E2 -7274.797} C_VEL
LIN {X 0,Y 475.159,Z 508.182,A -85,B 0,C 180,E1 -7276.093,E2 -7276.093} C_VEL
LIN {X 0,Y 474.665,Z 518.12,A -85,B 0,C 180,E1 -7277.572,E2 -7277.572} C_VEL
LIN {X 0,Y 474.423,Z 526.882,A -85,B 0,C 180,E1 -7279.113,E2 -7279.113} C_VEL
LIN {X 0,Y 474.13,Z 533.951,A -85,B 0,C 180,E1 -7280.616,E2 -7280.616} C_VEL
LIN {X 0,Y 474.004,Z 540.503,A -85,B 0,C 180,E1 -7282.332,E2 -7282.332} C_VEL
LIN {X 0,Y 473.988,Z 545.562,A -85,B 0,C 180,E1 -7284.043,E2 -7284.043} C_VEL
LIN {X 0,Y 473.935,Z 549.244,A -85,B 0,C 180,E1 -7285.748,E2 -7285.748} C_VEL
LIN {X 0,Y 473.927,Z 551.649,A -85,B 0,C 180,E1 -7287.45,E2 -7287.45} C_VEL
LIN {X 0,Y 473.866,Z 552.815,A -85,B 0,C 180,E1 -7289.15,E2 -7289.15} C_VEL
LIN {X 0,Y 473.875,Z 552.751,A -85,B 0,C 180,E1 -7290.85,E2 -7290.85} C_VEL
LIN {X 0,Y 473.948,Z 551.465,A -85,B 0,C 180,E1 -7292.55,E2 -7292.55} C_VEL
LIN {X 0,Y 474.035,Z 548.947,A -85,B 0,C 180,E1 -7294.251,E2 -7294.251} C_VEL
LIN {X 0,Y 474.027,Z 545.213,A -85,B 0,C 180,E1 -7295.957,E2 -7295.957} C_VEL
LIN {X 0,Y 474.039,Z 540.207,A -85,B 0,C 180,E1 -7297.668,E2 -7297.668} C_VEL
LIN {X 0,Y 474.154,Z 533.741,A -85,B 0,C 180,E1 -7299.384,E2 -7299.384} C_VEL
LIN {X 0,Y 474.43,Z 525.629,A -85,B 0,C 180,E1 -7301.103,E2 -7301.103} C_VEL
LIN {X 0,Y 474.751,Z 516.849,A -85,B 0,C 180,E1 -7302.631,E2 -7302.631} C_VEL
LIN {X 0,Y 475.23,Z 506.546,A -85,B 0,C 180,E1 -7304.124,E2 -7304.124} C_VEL
LIN {X 0,Y 475.781,Z 495.878,A -85,B 0,C 180,E1 -7305.42,E2 -7305.42} C_VEL
LIN {X 0,Y 476.498,Z 484.279,A -85,B 0,C 180,E1 -7306.604,E2 -7306.604} C_VEL
LIN {X 0,Y 477.169,Z 471.641,A -85,B 0,C 180,E1 -7307.685,E2 -7307.685} C_VEL
LIN {X 0,Y 477.863,Z 459.508,A -85,B 0,C 180,E1 -7308.545,E2 -7308.545} C_VEL
LIN {X 0,Y 478.586,Z 445.515,A -85,B 0,C 180,E1 -7309.35,E2 -7309.35} C_VEL
LIN {X 0,Y 479.179,Z 430.613,A -85,B 0,C 180,E1 -7310.018,E2 -7310.018} C_VEL
LIN {X 0,Y 479.613,Z 415.809,A -85,B 0,C 180,E1 -7310.505,E2 -7310.505} C_VEL
LIN {X 0,Y 477.672,Z 402.885,A -85,B 0,C 180,E1 -7310.889,E2 -7310.889} C_VEL
LIN {X 0,Y 475.651,Z 389.081,A -85,B 0,C 180,E1 -7311.224,E2 -7311.224} C_VEL
LIN {X 0,Y 476.347,Z 371.287,A -85,B 0,C 180,E1 -7314.401,E2 -7314.401} C_VEL
LIN {X 0,Y 477.221,Z 354.661,A -85,B 0,C 180,E1 -7317.558,E2 -7317.558} C_VEL
LIN {X 0,Y 478.399,Z 340.574,A -85,B 0,C 180,E1 -7320.453,E2 -7320.453} C_VEL
LIN {X 0,Y 479.783,Z 328.78,A -85,B 0,C 180,E1 -7323.128,E2 -7323.128} C_VEL
LIN {X 0,Y 481.313,Z 319.992,A -85,B 0,C 180,E1 -7325.353,E2 -7325.353} C_VEL
LIN {X 0,Y 481.101,Z 317.5,A -85,B 0,C 180,E1 -7326.118,E2 -7326.118} C_VEL
LIN {X 0,Y 479.507,Z 311.193,A -85,B 0,C 180,E1 -7328.473,E2 -7328.473} C_VEL
LIN {X 0,Y 478.196,Z 306.302,A -85,B 0,C 180,E1 -7330.84,E2 -7330.84} C_VEL
LIN {X 0,Y 477.491,Z 303.577,A -85,B 0,C 180,E1 -7332.614,E2 -7332.614} C_VEL
LIN {X 0,Y 476.78,Z 301.062,A -85,B 0,C 180,E1 -7335.036,E2 -7335.036} C_VEL
LIN {X 0,Y 476.361,Z 299.808,A -85,B 0,C 180,E1 -7337.534,E2 -7337.534} C_VEL
LIN {X 0,Y 476.172,Z 299.583,A -85,B 0,C 180,E1 -7340.129,E2 -7340.129} C_VEL
LIN {X 0,Y 476.117,Z 300.236,A -85,B 0,C 180,E1 -7342.854,E2 -7342.854} C_VEL
LIN {X 0,Y 475.953,Z 301.648,A -85,B 0,C 180,E1 -7345.867,E2 -7345.867} C_VEL
LIN {X 0,Y 475.584,Z 303.544,A -85,B 0,C 180,E1 -7348.993,E2 -7348.993} C_VEL
LIN {X 0,Y 475.436,Z 305.449,A -85,B 0,C 180,E1 -7351.769,E2 -7351.769} C_VEL
LIN {X 0,Y 475.295,Z 307.503,A -85,B 0,C 180,E1 -7354.608,E2 -7354.608} C_VEL
LIN {X 0,Y 475.141,Z 309.565,A -85,B 0,C 180,E1 -7357.383,E2 -7357.383} C_VEL
LIN {X 0,Y 475,Z 311.702,A -85,B 0,C 180,E1 -7360.105,E2 -7360.105} C_VEL
LIN {X 0,Y 474.857,Z 313.895,A -85,B 0,C 180,E1 -7362.782,E2 -7362.782} C_VEL
LIN {X 0,Y 474.885,Z 315.479,A -85,B 0,C 180,E1 -7364.452,E2 -7364.452} C_VEL
LIN {X 0,Y 478.546,Z 326.019,A -85,B 0,C 180,E1 -7364.999,E2 -7364.999} C_VEL
LIN {X 0,Y 478.357,Z 337.714,A -85,B 0,C 180,E1 -7365.537,E2 -7365.537} C_VEL
LIN {X 0,Y 477.855,Z 350.152,A -85,B 0,C 180,E1 -7366.276,E2 -7366.276} C_VEL
LIN {X 0,Y 477.279,Z 361.623,A -85,B 0,C 180,E1 -7367.136,E2 -7367.136} C_VEL
LIN {X 0,Y 476.818,Z 371.862,A -85,B 0,C 180,E1 -7368.091,E2 -7368.091} C_VEL
LIN {X 0,Y 476.365,Z 381.199,A -85,B 0,C 180,E1 -7369.158,E2 -7369.158} C_VEL
LIN {X 0,Y 475.852,Z 390.34,A -85,B 0,C 180,E1 -7370.436,E2 -7370.436} C_VEL
LIN {X 0,Y 475.411,Z 397.779,A -85,B 0,C 180,E1 -7371.734,E2 -7371.734} C_VEL
LIN {X 0,Y 475.113,Z 404.395,A -85,B 0,C 180,E1 -7373.204,E2 -7373.204} C_VEL
LIN {X 0,Y 474.814,Z 408.877,A -85,B 0,C 180,E1 -7374.479,E2 -7374.479} C_VEL
LIN {X 0,Y 474.607,Z 412.276,A -85,B 0,C 180,E1 -7375.754,E2 -7375.754} C_VEL
LIN {X 0,Y 474.643,Z 413.993,A -85,B 0,C 180,E1 -7376.605,E2 -7376.605} C_VEL
LIN {X 0,Y 474.479,Z 415.307,A -85,B 0,C 180,E1 -7377.453,E2 -7377.453} C_VEL
LIN {X 0,Y 474.395,Z 416.677,A -85,B 0,C 180,E1 -7379.151,E2 -7379.151} C_VEL
LIN {X 0,Y 474.377,Z 416.788,A -85,B 0,C 180,E1 -7380,E2 -7380} C_VEL
LIN {X 0,Y 474.381,Z 416.491,A -85,B 0,C 180,E1 -7380.849,E2 -7380.849} C_VEL
LIN {X 0,Y 474.274,Z 414.707,A -85,B 0,C 180,E1 -7382.548,E2 -7382.548} C_VEL
LIN {X 0,Y 474.352,Z 413.209,A -85,B 0,C 180,E1 -7383.398,E2 -7383.398} C_VEL
LIN {X 0,Y 474.522,Z 410.132,A -85,B 0,C 180,E1 -7384.673,E2 -7384.673} C_VEL
LIN {X 0,Y 474.585,Z 406.053,A -85,B 0,C 180,E1 -7385.95,E2 -7385.95} C_VEL
LIN {X 0,Y 474.89,Z 399.772,A -85,B 0,C 180,E1 -7387.452,E2 -7387.452} C_VEL
LIN {X 0,Y 475.172,Z 393.056,A -85,B 0,C 180,E1 -7388.72,E2 -7388.72} C_VEL
LIN {X 0,Y 475.436,Z 384.697,A -85,B 0,C 180,E1 -7390.003,E2 -7390.003} C_VEL
LIN {X 0,Y 475.866,Z 376.181,A -85,B 0,C 180,E1 -7391.069,E2 -7391.069} C_VEL
LIN {X 0,Y 476.307,Z 365.775,A -85,B 0,C 180,E1 -7392.138,E2 -7392.138} C_VEL
LIN {X 0,Y 476.738,Z 354.535,A -85,B 0,C 180,E1 -7393.072,E2 -7393.072} C_VEL
LIN {X 0,Y 477.156,Z 342.88,A -85,B 0,C 180,E1 -7393.848,E2 -7393.848} C_VEL
LIN {X 0,Y 477.519,Z 330.33,A -85,B 0,C 180,E1 -7394.49,E2 -7394.49} C_VEL
LIN {X 0,Y 477.461,Z 322.911,A -85,B 0,C 180,E1 -7394.798,E2 -7394.798} C_VEL
LIN {X 0,Y 474.076,Z 309.94,A -85,B 0,C 180,E1 -7395.325,E2 -7395.325} C_VEL
LIN {X 0,Y 474.074,Z 306.529,A -85,B 0,C 180,E1 -7398.417,E2 -7398.417} C_VEL
LIN {X 0,Y 474.078,Z 302.91,A -85,B 0,C 180,E1 -7401.754,E2 -7401.754} C_VEL
LIN {X 0,Y 474.109,Z 299.956,A -85,B 0,C 180,E1 -7404.523,E2 -7404.523} C_VEL
LIN {X 0,Y 474.134,Z 296.912,A -85,B 0,C 180,E1 -7407.355,E2 -7407.355} C_VEL
LIN {X 0,Y 474.143,Z 293.825,A -85,B 0,C 180,E1 -7410.263,E2 -7410.263} C_VEL
LIN {X 0,Y 474.205,Z 292.045,A -85,B 0,C 180,E1 -7412.245,E2 -7412.245} C_VEL
LIN {X 0,Y 474.539,Z 292.003,A -85,B 0,C 180,E1 -7415.456,E2 -7415.456} C_VEL
LIN {X 0,Y 474.613,Z 291.989,A -85,B 0,C 180,E1 -7418.457,E2 -7418.457} C_VEL
LIN {X 0,Y 474.63,Z 291.987,A -85,B 0,C 180,E1 -7420.959,E2 -7420.959} C_VEL
LIN {X 0,Y 474.607,Z 291.99,A -85,B 0,C 180,E1 -7424.105,E2 -7424.105} C_VEL
LIN {X 0,Y 474.57,Z 291.995,A -85,B 0,C 180,E1 -7427.06,E2 -7427.06} C_VEL
LIN {X 0,Y 474.525,Z 292.124,A -85,B 0,C 180,E1 -7429.332,E2 -7429.332} C_VEL
LIN {X 0,Y 474.586,Z 295.605,A -85,B 0,C 180,E1 -7431.708,E2 -7431.708} C_VEL
LIN {X 0,Y 474.52,Z 299.826,A -85,B 0,C 180,E1 -7434.716,E2 -7434.716} C_VEL
LIN {X 0,Y 474.486,Z 303.973,A -85,B 0,C 180,E1 -7437.776,E2 -7437.776} C_VEL
LIN {X 0,Y 474.399,Z 308.224,A -85,B 0,C 180,E1 -7440.934,E2 -7440.934} C_VEL
LIN {X 0,Y 474.323,Z 312.141,A -85,B 0,C 180,E1 -7443.744,E2 -7443.744} C_VEL
LIN {X 0,Y 474.291,Z 316.558,A -85,B 0,C 180,E1 -7446.739,E2 -7446.739} C_VEL
LIN {X 0,Y 474.267,Z 317.544,A -85,B 0,C 180,E1 -7447.381,E2 -7447.381} C_VEL
LIN {X 0,Y 474.273,Z 318.984,A -85,B 0,C 180,E1 -7447.803,E2 -7447.803} C_VEL
LIN {X 0,Y 474.302,Z 321.447,A -85,B 0,C 180,E1 -7448.156,E2 -7448.156} C_VEL
LIN {X 0,Y 474.35,Z 326.298,A -85,B 0,C 180,E1 -7448.563,E2 -7448.563} C_VEL
LIN {X 0,Y 474.359,Z 332.139,A -85,B 0,C 180,E1 -7448.849,E2 -7448.849} C_VEL
LIN {X 0,Y 474.097,Z 344.72,A -85,B 0,C 180,E1 -7449.255,E2 -7449.255} C_VEL
LIN {X 0,Y 473.554,Z 359.387,A -85,B 0,C 180,E1 -7449.836,E2 -7449.836} C_VEL
LIN {X 0,Y 473.005,Z 371.646,A -85,B 0,C 180,E1 -7450.469,E2 -7450.469} C_VEL
LIN {X 0,Y 472.274,Z 385.236,A -85,B 0,C 180,E1 -7451.34,E2 -7451.34} C_VEL
LIN {X 0,Y 471.486,Z 397.692,A -85,B 0,C 180,E1 -7452.319,E2 -7452.319} C_VEL
LIN {X 0,Y 470.599,Z 410.265,A -85,B 0,C 180,E1 -7453.516,E2 -7453.516} C_VEL
LIN {X 0,Y 469.784,Z 421.647,A -85,B 0,C 180,E1 -7454.823,E2 -7454.823} C_VEL
LIN {X 0,Y 468.965,Z 432.655,A -85,B 0,C 180,E1 -7456.347,E2 -7456.347} C_VEL
LIN {X 0,Y 468.379,Z 441.754,A -85,B 0,C 180,E1 -7457.873,E2 -7457.873} C_VEL
LIN {X 0,Y 467.915,Z 448.346,A -85,B 0,C 180,E1 -7459.178,E2 -7459.178} C_VEL
LIN {X 0,Y 467.487,Z 455.578,A -85,B 0,C 180,E1 -7460.918,E2 -7460.918} C_VEL
LIN {X 0,Y 467.174,Z 461.312,A -85,B 0,C 180,E1 -7462.653,E2 -7462.653} C_VEL
LIN {X 0,Y 467.008,Z 464.696,A -85,B 0,C 180,E1 -7463.953,E2 -7463.953} C_VEL
LIN {X 0,Y 466.897,Z 468.143,A -85,B 0,C 180,E1 -7465.683,E2 -7465.683} C_VEL
LIN {X 0,Y 466.824,Z 470.418,A -85,B 0,C 180,E1 -7467.411,E2 -7467.411} C_VEL
LIN {X 0,Y 466.655,Z 471.588,A -85,B 0,C 180,E1 -7469.137,E2 -7469.137} C_VEL
LIN {X 0,Y 466.654,Z 471.604,A -85,B 0,C 180,E1 -7470.863,E2 -7470.863} C_VEL
LIN {X 0,Y 466.824,Z 470.495,A -85,B 0,C 180,E1 -7472.588,E2 -7472.588} C_VEL
LIN {X 0,Y 466.897,Z 468.284,A -85,B 0,C 180,E1 -7474.316,E2 -7474.316} C_VEL
LIN {X 0,Y 467.005,Z 464.912,A -85,B 0,C 180,E1 -7476.047,E2 -7476.047} C_VEL
LIN {X 0,Y 467.24,Z 460.281,A -85,B 0,C 180,E1 -7477.78,E2 -7477.78} C_VEL
LIN {X 0,Y 467.549,Z 454.267,A -85,B 0,C 180,E1 -7479.517,E2 -7479.517} C_VEL
LIN {X 0,Y 468.028,Z 446.693,A -85,B 0,C 180,E1 -7481.257,E2 -7481.257} C_VEL
LIN {X 0,Y 468.554,Z 438.215,A -85,B 0,C 180,E1 -7482.849,E2 -7482.849} C_VEL
LIN {X 0,Y 469.285,Z 428.85,A -85,B 0,C 180,E1 -7484.306,E2 -7484.306} C_VEL
LIN {X 0,Y 470.037,Z 418.874,A -85,B 0,C 180,E1 -7485.613,E2 -7485.613} C_VEL
LIN {X 0,Y 470.843,Z 406.946,A -85,B 0,C 180,E1 -7486.919,E2 -7486.919} C_VEL
LIN {X 0,Y 471.692,Z 394.944,A -85,B 0,C 180,E1 -7488.009,E2 -7488.009} C_VEL
LIN {X 0,Y 472.468,Z 381.876,A -85,B 0,C 180,E1 -7488.989,E2 -7488.989} C_VEL
LIN {X 0,Y 473.224,Z 367.392,A -85,B 0,C 180,E1 -7489.86,E2 -7489.86} C_VEL
LIN {X 0,Y 473.792,Z 353.241,A -85,B 0,C 180,E1 -7490.524,E2 -7490.524} C_VEL
LIN {X 0,Y 474.047,Z 340.53,A -85,B 0,C 180,E1 -7490.978,E2 -7490.978} C_VEL
LIN {X 0,Y 469.865,Z 327.563,A -85,B 0,C 180,E1 -7491.525,E2 -7491.525} C_VEL
LIN {X 0,Y 467.277,Z 320.073,A -85,B 0,C 180,E1 -7491.814,E2 -7491.814} C_VEL
LIN {X 0,Y 467.272,Z 315.272,A -85,B 0,C 180,E1 -7494.906,E2 -7494.906} C_VEL
LIN {X 0,Y 467.343,Z 311.126,A -85,B 0,C 180,E1 -7497.787,E2 -7497.787} C_VEL
LIN {X 0,Y 467.39,Z 307.07,A -85,B 0,C 180,E1 -7500.747,E2 -7500.747} C_VEL
LIN {X 0,Y 467.458,Z 302.975,A -85,B 0,C 180,E1 -7503.799,E2 -7503.799} C_VEL
LIN {X 0,Y 467.522,Z 298.34,A -85,B 0,C 180,E1 -7507.182,E2 -7507.182} C_VEL
LIN {X 0,Y 467.533,Z 294.352,A -85,B 0,C 180,E1 -7509.947,E2 -7509.947} C_VEL
LIN {X 0,Y 467.492,Z 292.888,A -85,B 0,C 180,E1 -7511.017,E2 -7511.017} C_VEL
LIN {X 0,Y 467.546,Z 292.875,A -85,B 0,C 180,E1 -7513.82,E2 -7513.82} C_VEL
LIN {X 0,Y 467.557,Z 292.871,A -85,B 0,C 180,E1 -7516.256,E2 -7516.256} C_VEL
LIN {X 0,Y 467.578,Z 292.867,A -85,B 0,C 180,E1 -7518.723,E2 -7518.723} C_VEL
LIN {X 0,Y 467.563,Z 292.872,A -85,B 0,C 180,E1 -7521.955,E2 -7521.955} C_VEL
LIN {X 0,Y 467.566,Z 292.872,A -85,B 0,C 180,E1 -7525.167,E2 -7525.167} C_VEL
LIN {X 0,Y 467.582,Z 292.867,A -85,B 0,C 180,E1 -7528.26,E2 -7528.26} C_VEL
LIN {X 0,Y 467.542,Z 292.869,A -85,B 0,C 180,E1 -7531.248,E2 -7531.248} C_VEL
LIN {X 0,Y 467.578,Z 292.861,A -85,B 0,C 180,E1 -7534.401,E2 -7534.401} C_VEL
LIN {X 0,Y 467.576,Z 292.866,A -85,B 0,C 180,E1 -7536.996,E2 -7536.996} C_VEL
LIN {X 0,Y 467.621,Z 292.858,A -85,B 0,C 180,E1 -7539.777,E2 -7539.777} C_VEL
LIN {X 0,Y 467.589,Z 292.857,A -85,B 0,C 180,E1 -7542.506,E2 -7542.506} C_VEL
LIN {X 0,Y 467.61,Z 292.864,A -85,B 0,C 180,E1 -7545.196,E2 -7545.196} C_VEL
LIN {X 0,Y 467.657,Z 292.849,A -85,B 0,C 180,E1 -7547.854,E2 -7547.854} C_VEL
LIN {X 0,Y 467.664,Z 292.855,A -85,B 0,C 180,E1 -7551.357,E2 -7551.357} C_VEL
LIN {X 0,Y 467.71,Z 292.841,A -85,B 0,C 180,E1 -7553.962,E2 -7553.962} C_VEL
LIN {X 0,Y 467.858,Z 292.83,A -85,B 0,C 180,E1 -7557.417,E2 -7557.417} C_VEL
LIN {X 0,Y 467.883,Z 292.819,A -85,B 0,C 180,E1 -7560,E2 -7560} C_VEL
LIN {X 0,Y 467.848,Z 292.831,A -85,B 0,C 180,E1 -7562.583,E2 -7562.583} C_VEL
LIN {X 0,Y 467.717,Z 292.841,A -85,B 0,C 180,E1 -7566.038,E2 -7566.038} C_VEL
LIN {X 0,Y 467.671,Z 292.856,A -85,B 0,C 180,E1 -7568.643,E2 -7568.643} C_VEL
LIN {X 0,Y 467.657,Z 292.855,A -85,B 0,C 180,E1 -7572.145,E2 -7572.145} C_VEL
LIN {X 0,Y 467.648,Z 292.849,A -85,B 0,C 180,E1 -7575.885,E2 -7575.885} C_VEL
LIN {X 0,Y 467.622,Z 292.86,A -85,B 0,C 180,E1 -7579.308,E2 -7579.308} C_VEL
LIN {X 0,Y 467.534,Z 292.867,A -85,B 0,C 180,E1 -7582.074,E2 -7582.074} C_VEL
LIN {X 0,Y 467.567,Z 292.869,A -85,B 0,C 180,E1 -7584.889,E2 -7584.889} C_VEL
LIN {X 0,Y 467.578,Z 292.863,A -85,B 0,C 180,E1 -7587.772,E2 -7587.772} C_VEL
LIN {X 0,Y 467.568,Z 292.866,A -85,B 0,C 180,E1 -7591.045,E2 -7591.045} C_VEL
LIN {X 0,Y 467.587,Z 292.864,A -85,B 0,C 180,E1 -7594.242,E2 -7594.242} C_VEL
LIN {X 0,Y 467.541,Z 292.873,A -85,B 0,C 180,E1 -7597.185,E2 -7597.185} C_VEL
LIN {X 0,Y 467.573,Z 292.869,A -85,B 0,C 180,E1 -7600.265,E2 -7600.265} C_VEL
LIN {X 0,Y 467.586,Z 292.863,A -85,B 0,C 180,E1 -7602.567,E2 -7602.567} C_VEL
LIN {X 0,Y 467.564,Z 292.863,A -85,B 0,C 180,E1 -7605.052,E2 -7605.052} C_VEL
LIN {X 0,Y 467.566,Z 292.996,A -85,B 0,C 180,E1 -7607.631,E2 -7607.631} C_VEL
LIN {X 0,Y 470.453,Z 304.251,A -85,B 0,C 180,E1 -7610.639,E2 -7610.639} C_VEL
LIN {X 0,Y 473.359,Z 315.967,A -85,B 0,C 180,E1 -7613.567,E2 -7613.567} C_VEL
LIN {X 0,Y 474.13,Z 319.595,A -85,B 0,C 180,E1 -7614.423,E2 -7614.423} C_VEL
LIN {X 0,Y 472.672,Z 335.041,A -85,B 0,C 180,E1 -7617.638,E2 -7617.638} C_VEL
LIN {X 0,Y 471.336,Z 350.67,A -85,B 0,C 180,E1 -7620.769,E2 -7620.769} C_VEL
LIN {X 0,Y 470.183,Z 367.405,A -85,B 0,C 180,E1 -7624.013,E2 -7624.013} C_VEL
LIN {X 0,Y 469.198,Z 384.908,A -85,B 0,C 180,E1 -7627.313,E2 -7627.313} C_VEL
LIN {X 0,Y 468.912,Z 391.376,A -85,B 0,C 180,E1 -7628.515,E2 -7628.515} C_VEL
LIN {X 0,Y 471.612,Z 408.943,A -85,B 0,C 180,E1 -7628.969,E2 -7628.969} C_VEL
LIN {X 0,Y 472.922,Z 418.311,A -85,B 0,C 180,E1 -7629.286,E2 -7629.286} C_VEL
LIN {X 0,Y 472.374,Z 432.332,A -85,B 0,C 180,E1 -7629.78,E2 -7629.78} C_VEL
LIN {X 0,Y 471.744,Z 445.93,A -85,B 0,C 180,E1 -7630.415,E2 -7630.415} C_VEL
LIN {X 0,Y 471.031,Z 458.905,A -85,B 0,C 180,E1 -7631.177,E2 -7631.177} C_VEL
LIN {X 0,Y 470.202,Z 472.433,A -85,B 0,C 180,E1 -7632.157,E2 -7632.157} C_VEL
LIN {X 0,Y 469.513,Z 484.854,A -85,B 0,C 180,E1 -7633.254,E2 -7633.254} C_VEL
LIN {X 0,Y 468.72,Z 497.21,A -85,B 0,C 180,E1 -7634.565,E2 -7634.565} C_VEL
LIN {X 0,Y 468.159,Z 507.588,A -85,B 0,C 180,E1 -7635.881,E2 -7635.881} C_VEL
LIN {X 0,Y 467.61,Z 517.987,A -85,B 0,C 180,E1 -7637.457,E2 -7637.457} C_VEL
LIN {X 0,Y 467.331,Z 527.239,A -85,B 0,C 180,E1 -7639.165,E2 -7639.165} C_VEL
LIN {X 0,Y 467.015,Z 534.901,A -85,B 0,C 180,E1 -7640.909,E2 -7640.909} C_VEL
LIN {X 0,Y 466.92,Z 540.987,A -85,B 0,C 180,E1 -7642.65,E2 -7642.65} C_VEL
LIN {X 0,Y 466.939,Z 544.633,A -85,B 0,C 180,E1 -7643.952,E2 -7643.952} C_VEL
LIN {X 0,Y 466.885,Z 548.297,A -85,B 0,C 180,E1 -7645.684,E2 -7645.684} C_VEL
LIN {X 0,Y 466.882,Z 550.699,A -85,B 0,C 180,E1 -7647.412,E2 -7647.412} C_VEL
LIN {X 0,Y 466.828,Z 551.876,A -85,B 0,C 180,E1 -7649.138,E2 -7649.138} C_VEL
LIN {X 0,Y 466.828,Z 551.876,A -85,B 0,C 180,E1 -7650.863,E2 -7650.863} C_VEL
LIN {X 0,Y 466.887,Z 550.672,A -85,B 0,C 180,E1 -7652.588,E2 -7652.588} C_VEL
LIN {X 0,Y 466.978,Z 548.269,A -85,B 0,C 180,E1 -7654.316,E2 -7654.316} C_VEL
LIN {X 0,Y 466.952,Z 544.599,A -85,B 0,C 180,E1 -7656.048,E2 -7656.048} C_VEL
LIN {X 0,Y 466.953,Z 539.592,A -85,B 0,C 180,E1 -7657.785,E2 -7657.785} C_VEL
LIN {X 0,Y 467.064,Z 533.127,A -85,B 0,C 180,E1 -7659.528,E2 -7659.528} C_VEL
LIN {X 0,Y 467.363,Z 526.158,A -85,B 0,C 180,E1 -7661.054,E2 -7661.054} C_VEL
LIN {X 0,Y 467.648,Z 517.99,A -85,B 0,C 180,E1 -7662.543,E2 -7662.543} C_VEL
LIN {X 0,Y 468.172,Z 507.587,A -85,B 0,C 180,E1 -7664.119,E2 -7664.119} C_VEL
LIN {X 0,Y 468.734,Z 497.207,A -85,B 0,C 180,E1 -7665.435,E2 -7665.435} C_VEL
LIN {X 0,Y 469.494,Z 485.721,A -85,B 0,C 180,E1 -7666.658,E2 -7666.658} C_VEL
LIN {X 0,Y 470.162,Z 473.73,A -85,B 0,C 180,E1 -7667.732,E2 -7667.732} C_VEL
LIN {X 0,Y 470.961,Z 460.499,A -85,B 0,C 180,E1 -7668.714,E2 -7668.714} C_VEL
LIN {X 0,Y 471.71,Z 446.918,A -85,B 0,C 180,E1 -7669.53,E2 -7669.53} C_VEL
LIN {X 0,Y 472.372,Z 432.25,A -85,B 0,C 180,E1 -7670.223,E2 -7670.223} C_VEL
LIN {X 0,Y 472.91,Z 416.961,A -85,B 0,C 180,E1 -7670.756,E2 -7670.756} C_VEL
LIN {X 0,Y 471.06,Z 404.003,A -85,B 0,C 180,E1 -7671.165,E2 -7671.165} C_VEL
LIN {X 0,Y 468.968,Z 390.318,A -85,B 0,C 180,E1 -7671.497,E2 -7671.497} C_VEL
LIN {X 0,Y 468.639,Z 388.122,A -85,B 0,C 180,E1 -7671.56,E2 -7671.56} C_VEL
LIN {X 0,Y 469.346,Z 371.775,A -85,B 0,C 180,E1 -7674.555,E2 -7674.555} C_VEL
LIN {X 0,Y 470.263,Z 356.124,A -85,B 0,C 180,E1 -7677.6,E2 -7677.6} C_VEL
LIN {X 0,Y 471.47,Z 342.548,A -85,B 0,C 180,E1 -7680.453,E2 -7680.453} C_VEL
LIN {X 0,Y 473.046,Z 330.082,A -85,B 0,C 180,E1 -7683.347,E2 -7683.347} C_VEL
LIN {X 0,Y 474.556,Z 321.997,A -85,B 0,C 180,E1 -7685.459,E2 -7685.459} C_VEL
LIN {X 0,Y 474.62,Z 320.82,A -85,B 0,C 180,E1 -7685.811,E2 -7685.811} C_VEL
LIN {X 0,Y 473.116,Z 314.624,A -85,B 0,C 180,E1 -7688.066,E2 -7688.066} C_VEL
LIN {X 0,Y 471.693,Z 309.316,A -85,B 0,C 180,E1 -7690.547,E2 -7690.547} C_VEL
LIN {X 0,Y 471.01,Z 306.632,A -85,B 0,C 180,E1 -7692.18,E2 -7692.18} C_VEL
LIN {X 0,Y 470.169,Z 303.797,A -85,B 0,C 180,E1 -7694.632,E2 -7694.632} C_VEL
LIN {X 0,Y 469.662,Z 302.192,A -85,B 0,C 180,E1 -7697.159,E2 -7697.159} C_VEL
LIN {X 0,Y 469.419,Z 301.667,A -85,B 0,C 180,E1 -7699.779,E2 -7699.779} C_VEL
LIN {X 0,Y 469.288,Z 302.053,A -85,B 0,C 180,E1 -7702.535,E2 -7702.535} C_VEL
LIN {X 0,Y 469.065,Z 303.211,A -85,B 0,C 180,E1 -7705.494,E2 -7705.494} C_VEL
LIN {X 0,Y 468.729,Z 304.774,A -85,B 0,C 180,E1 -7708.347,E2 -7708.347} C_VEL
LIN {X 0,Y 468.516,Z 306.678,A -85,B 0,C 180,E1 -7711.314,E2 -7711.314} C_VEL
LIN {X 0,Y 468.354,Z 308.632,A -85,B 0,C 180,E1 -7714.204,E2 -7714.204} C_VEL
LIN {X 0,Y 468.199,Z 310.731,A -85,B 0,C 180,E1 -7717.028,E2 -7717.028} C_VEL
LIN {X 0,Y 468.052,Z 312.844,A -85,B 0,C 180,E1 -7719.797,E2 -7719.797} C_VEL
LIN {X 0,Y 467.891,Z 315.044,A -85,B 0,C 180,E1 -7722.518,E2 -7722.518} C_VEL
LIN {X 0,Y 467.897,Z 316.376,A -85,B 0,C 180,E1 -7724.114,E2 -7724.114} C_VEL
LIN {X 0,Y 471.623,Z 326.79,A -85,B 0,C 180,E1 -7724.69,E2 -7724.69} C_VEL
LIN {X 0,Y 472.037,Z 328.607,A -85,B 0,C 180,E1 -7724.787,E2 -7724.787} C_VEL
LIN {X 0,Y 471.59,Z 341.641,A -85,B 0,C 180,E1 -7725.425,E2 -7725.425} C_VEL
LIN {X 0,Y 471.071,Z 353.67,A -85,B 0,C 180,E1 -7726.19,E2 -7726.19} C_VEL
LIN {X 0,Y 470.434,Z 365.638,A -85,B 0,C 180,E1 -7727.16,E2 -7727.16} C_VEL
LIN {X 0,Y 469.859,Z 375.345,A -85,B 0,C 180,E1 -7728.131,E2 -7728.131} C_VEL
LIN {X 0,Y 469.437,Z 384.221,A -85,B 0,C 180,E1 -7729.214,E2 -7729.214} C_VEL
LIN {X 0,Y 468.83,Z 392.94,A -85,B 0,C 180,E1 -7730.509,E2 -7730.509} C_VEL
LIN {X 0,Y 468.493,Z 399.382,A -85,B 0,C 180,E1 -7731.687,E2 -7731.687} C_VEL
LIN {X 0,Y 468.166,Z 405.602,A -85,B 0,C 180,E1 -7733.103,E2 -7733.103} C_VEL
LIN {X 0,Y 467.859,Z 410.056,A -85,B 0,C 180,E1 -7734.397,E2 -7734.397} C_VEL
LIN {X 0,Y 467.623,Z 413.433,A -85,B 0,C 180,E1 -7735.69,E2 -7735.69} C_VEL
LIN {X 0,Y 467.67,Z 415.119,A -85,B 0,C 180,E1 -7736.554,E2 -7736.554} C_VEL
LIN {X 0,Y 467.498,Z 416.408,A -85,B 0,C 180,E1 -7737.415,E2 -7737.415} C_VEL
LIN {X 0,Y 467.382,Z 417.743,A -85,B 0,C 180,E1 -7739.139,E2 -7739.139} C_VEL
LIN {X 0,Y 467.362,Z 417.835,A -85,B 0,C 180,E1 -7740,E2 -7740} C_VEL
LIN {X 0,Y 467.367,Z 417.516,A -85,B 0,C 180,E1 -7740.862,E2 -7740.862} C_VEL
LIN {X 0,Y 467.25,Z 415.691,A -85,B 0,C 180,E1 -7742.586,E2 -7742.586} C_VEL
LIN {X 0,Y 467.33,Z 414.177,A -85,B 0,C 180,E1 -7743.449,E2 -7743.449} C_VEL
LIN {X 0,Y 467.515,Z 411.064,A -85,B 0,C 180,E1 -7744.743,E2 -7744.743} C_VEL
LIN {X 0,Y 467.592,Z 406.95,A -85,B 0,C 180,E1 -7746.039,E2 -7746.039} C_VEL
LIN {X 0,Y 467.897,Z 400.738,A -85,B 0,C 180,E1 -7747.541,E2 -7747.541} C_VEL
LIN {X 0,Y 468.218,Z 393.862,A -85,B 0,C 180,E1 -7748.85,E2 -7748.85} C_VEL
LIN {X 0,Y 468.498,Z 385.467,A -85,B 0,C 180,E1 -7750.152,E2 -7750.152} C_VEL
LIN {X 0,Y 468.959,Z 376.919,A -85,B 0,C 180,E1 -7751.234,E2 -7751.234} C_VEL
LIN {X 0,Y 469.428,Z 366.478,A -85,B 0,C 180,E1 -7752.318,E2 -7752.318} C_VEL
LIN {X 0,Y 469.864,Z 355.447,A -85,B 0,C 180,E1 -7753.249,E2 -7753.249} C_VEL
LIN {X 0,Y 470.318,Z 343.56,A -85,B 0,C 180,E1 -7754.053,E2 -7754.053} C_VEL
LIN {X 0,Y 470.702,Z 331.043,A -85,B 0,C 180,E1 -7754.704,E2 -7754.704} C_VEL
LIN {X 0,Y 470.685,Z 324.45,A -85,B 0,C 180,E1 -7754.985,E2 -7754.985} C_VEL
LIN {X 0,Y 467.018,Z 310.433,A -85,B 0,C 180,E1 -7755.591,E2 -7755.591} C_VEL
LIN {X 0,Y 467.019,Z 307.172,A -85,B 0,C 180,E1 -7758.546,E2 -7758.546} C_VEL
LIN {X 0,Y 467.059,Z 304.325,A -85,B 0,C 180,E1 -7761.17,E2 -7761.17} C_VEL
LIN {X 0,Y 467.037,Z 301.294,A -85,B 0,C 180,E1 -7763.973,E2 -7763.973} C_VEL
LIN {X 0,Y 467.039,Z 298.238,A -85,B 0,C 180,E1 -7766.836,E2 -7766.836} C_VEL
LIN {X 0,Y 467.082,Z 295.141,A -85,B 0,C 180,E1 -7769.771,E2 -7769.771} C_VEL
LIN {X 0,Y 467.099,Z 292.987,A -85,B 0,C 180,E1 -7771.777,E2 -7771.777} C_VEL
LIN {X 0,Y 467.433,Z 292.886,A -85,B 0,C 180,E1 -7774.844,E2 -7774.844} C_VEL
LIN {X 0,Y 467.565,Z 292.866,A -85,B 0,C 180,E1 -7778.045,E2 -7778.045} C_VEL
LIN {X 0,Y 467.581,Z 292.863,A -85,B 0,C 180,E1 -7781.277,E2 -7781.277} C_VEL
LIN {X 0,Y 467.551,Z 292.866,A -85,B 0,C 180,E1 -7783.82,E2 -7783.82} C_VEL
LIN {X 0,Y 467.547,Z 292.873,A -85,B 0,C 180,E1 -7786.254,E2 -7786.254} C_VEL
LIN {X 0,Y 467.511,Z 293.008,A -85,B 0,C 180,E1 -7789.233,E2 -7789.233} C_VEL
LIN {X 0,Y 467.543,Z 296.98,A -85,B 0,C 180,E1 -7791.953,E2 -7791.953} C_VEL
LIN {X 0,Y 467.467,Z 301.412,A -85,B 0,C 180,E1 -7795.159,E2 -7795.159} C_VEL
LIN {X 0,Y 467.42,Z 305.599,A -85,B 0,C 180,E1 -7798.247,E2 -7798.247} C_VEL
LIN {X 0,Y 467.345,Z 309.629,A -85,B 0,C 180,E1 -7801.235,E2 -7801.235} C_VEL
LIN {X 0,Y 467.288,Z 314.235,A -85,B 0,C 180,E1 -7804.475,E2 -7804.475} C_VEL
LIN {X 0,Y 467.247,Z 318.58,A -85,B 0,C 180,E1 -7807.355,E2 -7807.355} C_VEL
LIN {X 0,Y 467.282,Z 320.074,A -85,B 0,C 180,E1 -7808.29,E2 -7808.29} C_VEL
LIN {X 0,Y 472.843,Z 336.537,A -85,B 0,C 180,E1 -7808.935,E2 -7808.935} C_VEL
LIN {X 0,Y 474.145,Z 340.997,A -85,B 0,C 180,E1 -7809.134,E2 -7809.134} C_VEL
LIN {X 0,Y 474.097,Z 344.72,A -85,B 0,C 180,E1 -7809.255,E2 -7809.255} C_VEL
LIN {X 0,Y 473.232,Z 350.418,A -85,B 0,C 180,E1 -7809.42,E2 -7809.42} C_VEL
LIN {X 0,Y 470.154,Z 359.62,A -85,B 0,C 180,E1 -7809.677,E2 -7809.677} C_VEL
LIN {X 0,Y 467.117,Z 368.689,A -85,B 0,C 180,E1 -7810.003,E2 -7810.003} C_VEL
LIN {X 0,Y 466.281,Z 374.003,A -85,B 0,C 180,E1 -7810.282,E2 -7810.282} C_VEL
LIN {X 0,Y 465.464,Z 387.361,A -85,B 0,C 180,E1 -7811.171,E2 -7811.171} C_VEL
LIN {X 0,Y 464.686,Z 399.539,A -85,B 0,C 180,E1 -7812.165,E2 -7812.165} C_VEL
LIN {X 0,Y 463.746,Z 411.903,A -85,B 0,C 180,E1 -7813.378,E2 -7813.378} C_VEL
LIN {X 0,Y 462.941,Z 422.255,A -85,B 0,C 180,E1 -7814.593,E2 -7814.593} C_VEL
LIN {X 0,Y 462.194,Z 431.826,A -85,B 0,C 180,E1 -7815.919,E2 -7815.919} C_VEL
LIN {X 0,Y 461.541,Z 441.081,A -85,B 0,C 180,E1 -7817.45,E2 -7817.45} C_VEL
LIN {X 0,Y 460.948,Z 448.955,A -85,B 0,C 180,E1 -7819.013,E2 -7819.013} C_VEL
LIN {X 0,Y 460.503,Z 456.187,A -85,B 0,C 180,E1 -7820.779,E2 -7820.779} C_VEL
LIN {X 0,Y 460.153,Z 461.921,A -85,B 0,C 180,E1 -7822.54,E2 -7822.54} C_VEL
LIN {X 0,Y 459.968,Z 465.306,A -85,B 0,C 180,E1 -7823.86,E2 -7823.86} C_VEL
LIN {X 0,Y 459.85,Z 468.751,A -85,B 0,C 180,E1 -7825.617,E2 -7825.617} C_VEL
LIN {X 0,Y 459.771,Z 471.026,A -85,B 0,C 180,E1 -7827.371,E2 -7827.371} C_VEL
LIN {X 0,Y 459.586,Z 472.196,A -85,B 0,C 180,E1 -7829.124,E2 -7829.124} C_VEL
LIN {X 0,Y 459.586,Z 472.212,A -85,B 0,C 180,E1 -7830.876,E2 -7830.876} C_VEL
LIN {X 0,Y 459.772,Z 471.101,A -85,B 0,C 180,E1 -7832.628,E2 -7832.628} C_VEL
LIN {X 0,Y 459.849,Z 468.891,A -85,B 0,C 180,E1 -7834.382,E2 -7834.382} C_VEL
LIN {X 0,Y 459.965,Z 465.518,A -85,B 0,C 180,E1 -7836.14,E2 -7836.14} C_VEL
LIN {X 0,Y 460.223,Z 460.886,A -85,B 0,C 180,E1 -7837.899,E2 -7837.899} C_VEL
LIN {X 0,Y 460.551,Z 454.873,A -85,B 0,C 180,E1 -7839.663,E2 -7839.663} C_VEL
LIN {X 0,Y 461.082,Z 447.296,A -85,B 0,C 180,E1 -7841.429,E2 -7841.429} C_VEL
LIN {X 0,Y 461.626,Z 439.074,A -85,B 0,C 180,E1 -7843.001,E2 -7843.001} C_VEL
LIN {X 0,Y 462.431,Z 429.449,A -85,B 0,C 180,E1 -7844.523,E2 -7844.523} C_VEL
LIN {X 0,Y 463.208,Z 419.472,A -85,B 0,C 180,E1 -7845.849,E2 -7845.849} C_VEL
LIN {X 0,Y 464.058,Z 407.787,A -85,B 0,C 180,E1 -7847.149,E2 -7847.149} C_VEL
LIN {X 0,Y 464.967,Z 395.534,A -85,B 0,C 180,E1 -7848.278,E2 -7848.278} C_VEL
LIN {X 0,Y 465.784,Z 382.46,A -85,B 0,C 180,E1 -7849.272,E2 -7849.272} C_VEL
LIN {X 0,Y 466.586,Z 367.964,A -85,B 0,C 180,E1 -7850.155,E2 -7850.155} C_VEL
LIN {X 0,Y 467.169,Z 354.212,A -85,B 0,C 180,E1 -7850.811,E2 -7850.811} C_VEL
LIN {X 0,Y 467.421,Z 342.12,A -85,B 0,C 180,E1 -7851.254,E2 -7851.254} C_VEL
LIN {X 0,Y 463.231,Z 329.15,A -85,B 0,C 180,E1 -7851.825,E2 -7851.825} C_VEL
LIN {X 0,Y 460.253,Z 320.607,A -85,B 0,C 180,E1 -7852.172,E2 -7852.172} C_VEL
LIN {X 0,Y 460.254,Z 315.736,A -85,B 0,C 180,E1 -7855.312,E2 -7855.312} C_VEL
LIN {X 0,Y 460.305,Z 311.506,A -85,B 0,C 180,E1 -7858.249,E2 -7858.249} C_VEL
LIN {X 0,Y 460.378,Z 307.377,A -85,B 0,C 180,E1 -7861.267,E2 -7861.267} C_VEL
LIN {X 0,Y 460.45,Z 303.048,A -85,B 0,C 180,E1 -7864.49,E2 -7864.49} C_VEL
LIN {X 0,Y 460.514,Z 298.751,A -85,B 0,C 180,E1 -7867.622,E2 -7867.622} C_VEL
LIN {X 0,Y 460.512,Z 294.952,A -85,B 0,C 180,E1 -7870.265,E2 -7870.265} C_VEL
LIN {X 0,Y 460.462,Z 293.763,A -85,B 0,C 180,E1 -7871.162,E2 -7871.162} C_VEL
LIN {X 0,Y 460.515,Z 293.748,A -85,B 0,C 180,E1 -7874.589,E2 -7874.589} C_VEL
LIN {X 0,Y 460.523,Z 293.746,A -85,B 0,C 180,E1 -7877.818,E2 -7877.818} C_VEL
LIN {X 0,Y 460.532,Z 293.741,A -85,B 0,C 180,E1 -7881.104,E2 -7881.104} C_VEL
LIN {X 0,Y 460.512,Z 293.746,A -85,B 0,C 180,E1 -7884.554,E2 -7884.554} C_VEL
LIN {X 0,Y 460.531,Z 293.743,A -85,B 0,C 180,E1 -7887.715,E2 -7887.715} C_VEL
LIN {X 0,Y 460.519,Z 293.745,A -85,B 0,C 180,E1 -7890.767,E2 -7890.767} C_VEL
LIN {X 0,Y 460.535,Z 293.739,A -85,B 0,C 180,E1 -7894.207,E2 -7894.207} C_VEL
LIN {X 0,Y 460.511,Z 293.741,A -85,B 0,C 180,E1 -7897.571,E2 -7897.571} C_VEL
LIN {X 0,Y 460.567,Z 293.743,A -85,B 0,C 180,E1 -7900.384,E2 -7900.384} C_VEL
LIN {X 0,Y 460.605,Z 293.732,A -85,B 0,C 180,E1 -7904.059,E2 -7904.059} C_VEL
LIN {X 0,Y 460.61,Z 293.727,A -85,B 0,C 180,E1 -7907.666,E2 -7907.666} C_VEL
LIN {X 0,Y 460.616,Z 293.733,A -85,B 0,C 180,E1 -7911.224,E2 -7911.224} C_VEL
LIN {X 0,Y 460.675,Z 293.717,A -85,B 0,C 180,E1 -7913.87,E2 -7913.87} C_VEL
LIN {X 0,Y 460.798,Z 293.71,A -85,B 0,C 180,E1 -7917.377,E2 -7917.377} C_VEL
LIN {X 0,Y 460.853,Z 293.694,A -85,B 0,C 180,E1 -7920,E2 -7920} C_VEL
LIN {X 0,Y 460.788,Z 293.711,A -85,B 0,C 180,E1 -7922.622,E2 -7922.622} C_VEL
LIN {X 0,Y 460.684,Z 293.717,A -85,B 0,C 180,E1 -7926.13,E2 -7926.13} C_VEL
LIN {X 0,Y 460.621,Z 293.733,A -85,B 0,C 180,E1 -7928.776,E2 -7928.776} C_VEL
LIN {X 0,Y 460.61,Z 293.733,A -85,B 0,C 180,E1 -7932.334,E2 -7932.334} C_VEL
LIN {X 0,Y 460.6,Z 293.726,A -85,B 0,C 180,E1 -7935.997,E2 -7935.997} C_VEL
LIN {X 0,Y 460.568,Z 293.739,A -85,B 0,C 180,E1 -7939.615,E2 -7939.615} C_VEL
LIN {X 0,Y 460.51,Z 293.743,A -85,B 0,C 180,E1 -7942.429,E2 -7942.429} C_VEL
LIN {X 0,Y 460.534,Z 293.738,A -85,B 0,C 180,E1 -7945.793,E2 -7945.793} C_VEL
LIN {X 0,Y 460.525,Z 293.744,A -85,B 0,C 180,E1 -7948.235,E2 -7948.235} C_VEL
LIN {X 0,Y 460.52,Z 293.745,A -85,B 0,C 180,E1 -7951.283,E2 -7951.283} C_VEL
LIN {X 0,Y 460.53,Z 293.743,A -85,B 0,C 180,E1 -7954.505,E2 -7954.505} C_VEL
LIN {X 0,Y 460.497,Z 293.748,A -85,B 0,C 180,E1 -7957.623,E2 -7957.623} C_VEL
LIN {X 0,Y 460.538,Z 293.746,A -85,B 0,C 180,E1 -7960.269,E2 -7960.269} C_VEL
LIN {X 0,Y 460.498,Z 293.745,A -85,B 0,C 180,E1 -7963.375,E2 -7963.375} C_VEL
LIN {X 0,Y 460.502,Z 293.743,A -85,B 0,C 180,E1 -7966.625,E2 -7966.625} C_VEL
LIN {X 0,Y 460.492,Z 293.747,A -85,B 0,C 180,E1 -7967.102,E2 -7967.102} C_VEL
LIN {X 0,Y 463.125,Z 304.107,A -85,B 0,C 180,E1 -7969.939,E2 -7969.939} C_VEL
LIN {X 0,Y 466.153,Z 316.133,A -85,B 0,C 180,E1 -7973.04,E2 -7973.04} C_VEL
LIN {X 0,Y 467.312,Z 321.338,A -85,B 0,C 180,E1 -7974.303,E2 -7974.303} C_VEL
LIN {X 0,Y 465.849,Z 336.291,A -85,B 0,C 180,E1 -7977.463,E2 -7977.463} C_VEL
LIN {X 0,Y 464.37,Z 352.578,A -85,B 0,C 180,E1 -7980.785,E2 -7980.785} C_VEL
LIN {X 0,Y 463.204,Z 368.292,A -85,B 0,C 180,E1 -7983.896,E2 -7983.896} C_VEL
LIN {X 0,Y 462.199,Z 385.396,A -85,B 0,C 180,E1 -7987.186,E2 -7987.186} C_VEL
LIN {X 0,Y 461.918,Z 390.538,A -85,B 0,C 180,E1 -7988.161,E2 -7988.161} C_VEL
LIN {X 0,Y 464.556,Z 406.807,A -85,B 0,C 180,E1 -7988.594,E2 -7988.594} C_VEL
LIN {X 0,Y 466.226,Z 418.962,A -85,B 0,C 180,E1 -7989.012,E2 -7989.012} C_VEL
LIN {X 0,Y 465.611,Z 433.495,A -85,B 0,C 180,E1 -7989.55,E2 -7989.55} C_VEL
LIN {X 0,Y 464.886,Z 447.338,A -85,B 0,C 180,E1 -7990.229,E2 -7990.229} C_VEL
LIN {X 0,Y 464.016,Z 461.497,A -85,B 0,C 180,E1 -7991.111,E2 -7991.111} C_VEL
LIN {X 0,Y 463.196,Z 474.442,A -85,B 0,C 180,E1 -7992.107,E2 -7992.107} C_VEL
LIN {X 0,Y 462.461,Z 486.414,A -85,B 0,C 180,E1 -7993.217,E2 -7993.217} C_VEL
LIN {X 0,Y 461.662,Z 498.409,A -85,B 0,C 180,E1 -7994.55,E2 -7994.55} C_VEL
LIN {X 0,Y 461.08,Z 508.508,A -85,B 0,C 180,E1 -7995.885,E2 -7995.885} C_VEL
LIN {X 0,Y 460.522,Z 518.506,A -85,B 0,C 180,E1 -7997.462,E2 -7997.462} C_VEL
LIN {X 0,Y 460.261,Z 526.614,A -85,B 0,C 180,E1 -7998.997,E2 -7998.997} C_VEL
LIN {X 0,Y 459.928,Z 534.282,A -85,B 0,C 180,E1 -8000.767,E2 -8000.767} C_VEL
LIN {X 0,Y 459.839,Z 540.382,A -85,B 0,C 180,E1 -8002.536,E2 -8002.536} C_VEL
LIN {X 0,Y 459.847,Z 543.992,A -85,B 0,C 180,E1 -8003.859,E2 -8003.859} C_VEL
LIN {X 0,Y 459.798,Z 547.656,A -85,B 0,C 180,E1 -8005.617,E2 -8005.617} C_VEL
LIN {X 0,Y 459.823,Z 550.07,A -85,B 0,C 180,E1 -8007.372,E2 -8007.372} C_VEL
LIN {X 0,Y 459.754,Z 551.267,A -85,B 0,C 180,E1 -8009.124,E2 -8009.124} C_VEL
LIN {X 0,Y 459.754,Z 551.268,A -85,B 0,C 180,E1 -8010.876,E2 -8010.876} C_VEL
LIN {X 0,Y 459.828,Z 550.064,A -85,B 0,C 180,E1 -8012.628,E2 -8012.628} C_VEL
LIN {X 0,Y 459.886,Z 547.658,A -85,B 0,C 180,E1 -8014.382,E2 -8014.382} C_VEL
LIN {X 0,Y 459.861,Z 543.988,A -85,B 0,C 180,E1 -8016.141,E2 -8016.141} C_VEL
LIN {X 0,Y 459.869,Z 538.98,A -85,B 0,C 180,E1 -8017.906,E2 -8017.906} C_VEL
LIN {X 0,Y 459.987,Z 532.513,A -85,B 0,C 180,E1 -8019.676,E2 -8019.676} C_VEL
LIN {X 0,Y 460.27,Z 525.54,A -85,B 0,C 180,E1 -8021.226,E2 -8021.226} C_VEL
LIN {X 0,Y 460.656,Z 515.875,A -85,B 0,C 180,E1 -8022.983,E2 -8022.983} C_VEL
LIN {X 0,Y 461.161,Z 506.971,A -85,B 0,C 180,E1 -8024.339,E2 -8024.339} C_VEL
LIN {X 0,Y 461.782,Z 496.592,A -85,B 0,C 180,E1 -8025.673,E2 -8025.673} C_VEL
LIN {X 0,Y 462.621,Z 484.451,A -85,B 0,C 180,E1 -8026.981,E2 -8026.981} C_VEL
LIN {X 0,Y 463.397,Z 471.816,A -85,B 0,C 180,E1 -8028.114,E2 -8028.114} C_VEL
LIN {X 0,Y 464.253,Z 458.3,A -85,B 0,C 180,E1 -8029.109,E2 -8029.109} C_VEL
LIN {X 0,Y 465.165,Z 443.295,A -85,B 0,C 180,E1 -8029.989,E2 -8029.989} C_VEL
LIN {X 0,Y 465.845,Z 429.001,A -85,B 0,C 180,E1 -8030.637,E2 -8030.637} C_VEL
LIN {X 0,Y 466.099,Z 417.494,A -85,B 0,C 180,E1 -8031.038,E2 -8031.038} C_VEL
LIN {X 0,Y 464.418,Z 404.69,A -85,B 0,C 180,E1 -8031.459,E2 -8031.459} C_VEL
LIN {X 0,Y 462.048,Z 389.61,A -85,B 0,C 180,E1 -8031.839,E2 -8031.839} C_VEL
LIN {X 0,Y 461.678,Z 387.281,A -85,B 0,C 180,E1 -8031.896,E2 -8031.896} C_VEL
LIN {X 0,Y 462.481,Z 369.879,A -85,B 0,C 180,E1 -8035.182,E2 -8035.182} C_VEL
LIN {X 0,Y 463.427,Z 355.695,A -85,B 0,C 180,E1 -8038.043,E2 -8038.043} C_VEL
LIN {X 0,Y 464.608,Z 343.82,A -85,B 0,C 180,E1 -8040.615,E2 -8040.615} C_VEL
LIN {X 0,Y 466.54,Z 330.259,A -85,B 0,C 180,E1 -8043.875,E2 -8043.875} C_VEL
LIN {X 0,Y 467.847,Z 323.252,A -85,B 0,C 180,E1 -8045.788,E2 -8045.788} C_VEL
LIN {X 0,Y 466.751,Z 318.275,A -85,B 0,C 180,E1 -8047.576,E2 -8047.576} C_VEL
LIN {X 0,Y 465.539,Z 313.505,A -85,B 0,C 180,E1 -8049.653,E2 -8049.653} C_VEL
LIN {X 0,Y 464.369,Z 309.168,A -85,B 0,C 180,E1 -8052.133,E2 -8052.133} C_VEL
LIN {X 0,Y 463.534,Z 306.273,A -85,B 0,C 180,E1 -8054.553,E2 -8054.553} C_VEL
LIN {X 0,Y 462.985,Z 304.598,A -85,B 0,C 180,E1 -8056.915,E2 -8056.915} C_VEL
LIN {X 0,Y 462.674,Z 303.836,A -85,B 0,C 180,E1 -8059.42,E2 -8059.42} C_VEL
LIN {X 0,Y 462.474,Z 304.022,A -85,B 0,C 180,E1 -8062.565,E2 -8062.565} C_VEL
LIN {X 0,Y 462.159,Z 305.148,A -85,B 0,C 180,E1 -8065.761,E2 -8065.761} C_VEL
LIN {X 0,Y 461.791,Z 306.746,A -85,B 0,C 180,E1 -8068.839,E2 -8068.839} C_VEL
LIN {X 0,Y 461.53,Z 308.713,A -85,B 0,C 180,E1 -8072.032,E2 -8072.032} C_VEL
LIN {X 0,Y 461.38,Z 310.543,A -85,B 0,C 180,E1 -8074.754,E2 -8074.754} C_VEL
LIN {X 0,Y 461.2,Z 312.62,A -85,B 0,C 180,E1 -8077.607,E2 -8077.607} C_VEL
LIN {X 0,Y 461.055,Z 314.727,A -85,B 0,C 180,E1 -8080.406,E2 -8080.406} C_VEL
LIN {X 0,Y 460.934,Z 317.456,A -85,B 0,C 180,E1 -8083.77,E2 -8083.77} C_VEL
LIN {X 0,Y 465.437,Z 330.164,A -85,B 0,C 180,E1 -8084.51,E2 -8084.51} C_VEL
LIN {X 0,Y 464.896,Z 343.842,A -85,B 0,C 180,E1 -8085.209,E2 -8085.209} C_VEL
LIN {X 0,Y 464.349,Z 355.485,A -85,B 0,C 180,E1 -8085.986,E2 -8085.986} C_VEL
LIN {X 0,Y 463.681,Z 367.273,A -85,B 0,C 180,E1 -8086.97,E2 -8086.97} C_VEL
LIN {X 0,Y 463.072,Z 376.876,A -85,B 0,C 180,E1 -8087.955,E2 -8087.955} C_VEL
LIN {X 0,Y 462.615,Z 385.672,A -85,B 0,C 180,E1 -8089.053,E2 -8089.053} C_VEL
LIN {X 0,Y 461.964,Z 394.286,A -85,B 0,C 180,E1 -8090.367,E2 -8090.367} C_VEL
LIN {X 0,Y 461.504,Z 401.941,A -85,B 0,C 180,E1 -8091.832,E2 -8091.832} C_VEL
LIN {X 0,Y 461.22,Z 406.807,A -85,B 0,C 180,E1 -8092.998,E2 -8092.998} C_VEL
LIN {X 0,Y 460.901,Z 411.233,A -85,B 0,C 180,E1 -8094.312,E2 -8094.312} C_VEL
LIN {X 0,Y 460.637,Z 414.584,A -85,B 0,C 180,E1 -8095.625,E2 -8095.625} C_VEL
LIN {X 0,Y 460.692,Z 416.254,A -85,B 0,C 180,E1 -8096.502,E2 -8096.502} C_VEL
LIN {X 0,Y 460.515,Z 417.521,A -85,B 0,C 180,E1 -8097.376,E2 -8097.376} C_VEL
LIN {X 0,Y 460.368,Z 418.823,A -85,B 0,C 180,E1 -8099.125,E2 -8099.125} C_VEL
LIN {X 0,Y 460.346,Z 418.892,A -85,B 0,C 180,E1 -8100,E2 -8100} C_VEL
LIN {X 0,Y 460.352,Z 418.547,A -85,B 0,C 180,E1 -8100.875,E2 -8100.875} C_VEL
LIN {X 0,Y 460.227,Z 416.682,A -85,B 0,C 180,E1 -8102.626,E2 -8102.626} C_VEL
LIN {X 0,Y 460.308,Z 415.135,A -85,B 0,C 180,E1 -8103.501,E2 -8103.501} C_VEL
LIN {X 0,Y 460.509,Z 411.983,A -85,B 0,C 180,E1 -8104.815,E2 -8104.815} C_VEL
LIN {X 0,Y 460.601,Z 407.825,A -85,B 0,C 180,E1 -8106.131,E2 -8106.131} C_VEL
LIN {X 0,Y 460.928,Z 401.566,A -85,B 0,C 180,E1 -8107.653,E2 -8107.653} C_VEL
LIN {X 0,Y 461.269,Z 394.632,A -85,B 0,C 180,E1 -8108.985,E2 -8108.985} C_VEL
LIN {X 0,Y 461.563,Z 386.192,A -85,B 0,C 180,E1 -8110.306,E2 -8110.306} C_VEL
LIN {X 0,Y 462.053,Z 377.595,A -85,B 0,C 180,E1 -8111.405,E2 -8111.405} C_VEL
LIN {X 0,Y 462.542,Z 367.101,A -85,B 0,C 180,E1 -8112.505,E2 -8112.505} C_VEL
LIN {X 0,Y 463.061,Z 354.986,A -85,B 0,C 180,E1 -8113.53,E2 -8113.53} C_VEL
LIN {X 0,Y 463.466,Z 344.121,A -85,B 0,C 180,E1 -8114.266,E2 -8114.266} C_VEL
LIN {X 0,Y 463.882,Z 331.594,A -85,B 0,C 180,E1 -8114.925,E2 -8114.925} C_VEL
LIN {X 0,Y 463.818,Z 325.678,A -85,B 0,C 180,E1 -8115.185,E2 -8115.185} C_VEL
LIN {X 0,Y 460.113,Z 311.935,A -85,B 0,C 180,E1 -8115.783,E2 -8115.783} C_VEL
LIN {X 0,Y 459.959,Z 310.964,A -85,B 0,C 180,E1 -8115.836,E2 -8115.836} C_VEL
LIN {X 0,Y 459.962,Z 307.776,A -85,B 0,C 180,E1 -8118.716,E2 -8118.716} C_VEL
LIN {X 0,Y 459.982,Z 304.728,A -85,B 0,C 180,E1 -8121.512,E2 -8121.512} C_VEL
LIN {X 0,Y 460.002,Z 301.66,A -85,B 0,C 180,E1 -8124.363,E2 -8124.363} C_VEL
LIN {X 0,Y 460.025,Z 298.206,A -85,B 0,C 180,E1 -8127.613,E2 -8127.613} C_VEL
LIN {X 0,Y 460.029,Z 295.373,A -85,B 0,C 180,E1 -8130.275,E2 -8130.275} C_VEL
LIN {X 0,Y 460.031,Z 294.291,A -85,B 0,C 180,E1 -8131.294,E2 -8131.294} C_VEL
LIN {X 0,Y 460.17,Z 293.793,A -85,B 0,C 180,E1 -8132.86,E2 -8132.86} C_VEL
LIN {X 0,Y 460.434,Z 293.76,A -85,B 0,C 180,E1 -8135.453,E2 -8135.453} C_VEL
LIN {X 0,Y 460.547,Z 293.744,A -85,B 0,C 180,E1 -8138.897,E2 -8138.897} C_VEL
LIN {X 0,Y 460.526,Z 293.742,A -85,B 0,C 180,E1 -8142.181,E2 -8142.181} C_VEL
LIN {X 0,Y 460.513,Z 293.744,A -85,B 0,C 180,E1 -8145.411,E2 -8145.411} C_VEL
LIN {X 0,Y 460.472,Z 293.755,A -85,B 0,C 180,E1 -8148.982,E2 -8148.982} C_VEL
LIN {X 0,Y 460.527,Z 297.029,A -85,B 0,C 180,E1 -8151.267,E2 -8151.267} C_VEL
LIN {X 0,Y 460.473,Z 301.585,A -85,B 0,C 180,E1 -8154.551,E2 -8154.551} C_VEL
LIN {X 0,Y 460.393,Z 305.875,A -85,B 0,C 180,E1 -8157.704,E2 -8157.704} C_VEL
LIN {X 0,Y 460.358,Z 309.983,A -85,B 0,C 180,E1 -8160.756,E2 -8160.756} C_VEL
LIN {X 0,Y 460.273,Z 314.162,A -85,B 0,C 180,E1 -8163.717,E2 -8163.717} C_VEL
LIN {X 0,Y 460.262,Z 318.492,A -85,B 0,C 180,E1 -8166.608,E2 -8166.608} C_VEL
LIN {X 0,Y 460.271,Z 320.622,A -85,B 0,C 180,E1 -8167.936,E2 -8167.936} C_VEL
LIN {X 0,Y 465.934,Z 337.221,A -85,B 0,C 180,E1 -8168.61,E2 -8168.61} C_VEL
LIN {X 0,Y 467.529,Z 343.115,A -85,B 0,C 180,E1 -8168.877,E2 -8168.877} C_VEL
LIN {X 0,Y 467.026,Z 358.315,A -85,B 0,C 180,E1 -8169.465,E2 -8169.465} C_VEL
LIN {X 0,Y 466.344,Z 372.239,A -85,B 0,C 180,E1 -8170.179,E2 -8170.179} C_VEL
LIN {X 0,Y 466.281,Z 374.003,A -85,B 0,C 180,E1 -8170.282,E2 -8170.282} C_VEL
LIN {X 0,Y 465.412,Z 379.327,A -85,B 0,C 180,E1 -8170.58,E2 -8170.58} C_VEL
LIN {X 0,Y 462.147,Z 387.908,A -85,B 0,C 180,E1 -8171.048,E2 -8171.048} C_VEL
LIN {X 0,Y 458.847,Z 396.255,A -85,B 0,C 180,E1 -8171.577,E2 -8171.577} C_VEL
LIN {X 0,Y 457.899,Z 401.081,A -85,B 0,C 180,E1 -8171.979,E2 -8171.979} C_VEL
LIN {X 0,Y 456.969,Z 412.507,A -85,B 0,C 180,E1 -8173.124,E2 -8173.124} C_VEL
LIN {X 0,Y 456.113,Z 422.861,A -85,B 0,C 180,E1 -8174.356,E2 -8174.356} C_VEL
LIN {X 0,Y 455.332,Z 432.433,A -85,B 0,C 180,E1 -8175.702,E2 -8175.702} C_VEL
LIN {X 0,Y 454.617,Z 441.793,A -85,B 0,C 180,E1 -8177.276,E2 -8177.276} C_VEL
LIN {X 0,Y 453.997,Z 449.564,A -85,B 0,C 180,E1 -8178.842,E2 -8178.842} C_VEL
LIN {X 0,Y 453.501,Z 456.796,A -85,B 0,C 180,E1 -8180.635,E2 -8180.635} C_VEL
LIN {X 0,Y 453.125,Z 462.53,A -85,B 0,C 180,E1 -8182.424,E2 -8182.424} C_VEL
LIN {X 0,Y 452.931,Z 465.914,A -85,B 0,C 180,E1 -8183.764,E2 -8183.764} C_VEL
LIN {X 0,Y 452.803,Z 469.359,A -85,B 0,C 180,E1 -8185.549,E2 -8185.549} C_VEL
LIN {X 0,Y 452.721,Z 471.633,A -85,B 0,C 180,E1 -8187.33,E2 -8187.33} C_VEL
LIN {X 0,Y 452.52,Z 472.804,A -85,B 0,C 180,E1 -8189.11,E2 -8189.11} C_VEL
LIN {X 0,Y 452.52,Z 472.819,A -85,B 0,C 180,E1 -8190.89,E2 -8190.89} C_VEL
LIN {X 0,Y 452.722,Z 471.707,A -85,B 0,C 180,E1 -8192.669,E2 -8192.669} C_VEL
LIN {X 0,Y 452.803,Z 469.497,A -85,B 0,C 180,E1 -8194.451,E2 -8194.451} C_VEL
LIN {X 0,Y 452.928,Z 466.125,A -85,B 0,C 180,E1 -8196.235,E2 -8196.235} C_VEL
LIN {X 0,Y 453.204,Z 461.493,A -85,B 0,C 180,E1 -8198.023,E2 -8198.023} C_VEL
LIN {X 0,Y 453.562,Z 455.479,A -85,B 0,C 180,E1 -8199.814,E2 -8199.814} C_VEL
LIN {X 0,Y 454.143,Z 447.9,A -85,B 0,C 180,E1 -8201.606,E2 -8201.606} C_VEL
LIN {X 0,Y 454.701,Z 439.938,A -85,B 0,C 180,E1 -8203.157,E2 -8203.157} C_VEL
LIN {X 0,Y 455.576,Z 430.049,A -85,B 0,C 180,E1 -8204.746,E2 -8204.746} C_VEL
LIN {X 0,Y 456.4,Z 420.07,A -85,B 0,C 180,E1 -8206.092,E2 -8206.092} C_VEL
LIN {X 0,Y 457.277,Z 408.619,A -85,B 0,C 180,E1 -8207.387,E2 -8207.387} C_VEL
LIN {X 0,Y 458.249,Z 396.124,A -85,B 0,C 180,E1 -8208.556,E2 -8208.556} C_VEL
LIN {X 0,Y 459.133,Z 383.042,A -85,B 0,C 180,E1 -8209.563,E2 -8209.563} C_VEL
LIN {X 0,Y 459.968,Z 368.536,A -85,B 0,C 180,E1 -8210.457,E2 -8210.457} C_VEL
LIN {X 0,Y 460.6,Z 353.476,A -85,B 0,C 180,E1 -8211.175,E2 -8211.175} C_VEL
LIN {X 0,Y 460.865,Z 343.882,A -85,B 0,C 180,E1 -8211.53,E2 -8211.53} C_VEL
LIN {X 0,Y 456.599,Z 330.651,A -85,B 0,C 180,E1 -8212.137,E2 -8212.137} C_VEL
LIN {X 0,Y 453.252,Z 321.177,A -85,B 0,C 180,E1 -8212.52,E2 -8212.52} C_VEL
LIN {X 0,Y 453.251,Z 315.899,A -85,B 0,C 180,E1 -8215.929,E2 -8215.929} C_VEL
LIN {X 0,Y 453.3,Z 311.887,A -85,B 0,C 180,E1 -8218.726,E2 -8218.726} C_VEL
LIN {X 0,Y 453.351,Z 307.684,A -85,B 0,C 180,E1 -8221.808,E2 -8221.808} C_VEL
LIN {X 0,Y 453.43,Z 303.39,A -85,B 0,C 180,E1 -8224.994,E2 -8224.994} C_VEL
LIN {X 0,Y 453.5,Z 298.838,A -85,B 0,C 180,E1 -8228.308,E2 -8228.308} C_VEL
LIN {X 0,Y 453.43,Z 294.638,A -85,B 0,C 180,E1 -8231.351,E2 -8231.351} C_VEL
LIN {X 0,Y 453.485,Z 294.624,A -85,B 0,C 180,E1 -8234.529,E2 -8234.529} C_VEL
LIN {X 0,Y 453.48,Z 294.625,A -85,B 0,C 180,E1 -8238.209,E2 -8238.209} C_VEL
LIN {X 0,Y 453.47,Z 294.621,A -85,B 0,C 180,E1 -8240.797,E2 -8240.797} C_VEL
LIN {X 0,Y 453.455,Z 294.626,A -85,B 0,C 180,E1 -8243.917,E2 -8243.917} C_VEL
LIN {X 0,Y 453.483,Z 294.622,A -85,B 0,C 180,E1 -8247.151,E2 -8247.151} C_VEL
LIN {X 0,Y 453.461,Z 294.621,A -85,B 0,C 180,E1 -8250.267,E2 -8250.267} C_VEL
LIN {X 0,Y 453.442,Z 294.625,A -85,B 0,C 180,E1 -8253.29,E2 -8253.29} C_VEL
LIN {X 0,Y 453.494,Z 294.62,A -85,B 0,C 180,E1 -8256.238,E2 -8256.238} C_VEL
LIN {X 0,Y 453.482,Z 294.619,A -85,B 0,C 180,E1 -8259.118,E2 -8259.118} C_VEL
LIN {X 0,Y 453.498,Z 294.617,A -85,B 0,C 180,E1 -8261.944,E2 -8261.944} C_VEL
LIN {X 0,Y 453.542,Z 294.612,A -85,B 0,C 180,E1 -8264.726,E2 -8264.726} C_VEL
LIN {X 0,Y 453.56,Z 294.604,A -85,B 0,C 180,E1 -8268.379,E2 -8268.379} C_VEL
LIN {X 0,Y 453.583,Z 294.609,A -85,B 0,C 180,E1 -8271.086,E2 -8271.086} C_VEL
LIN {X 0,Y 453.642,Z 294.593,A -85,B 0,C 180,E1 -8273.774,E2 -8273.774} C_VEL
LIN {X 0,Y 453.742,Z 294.589,A -85,B 0,C 180,E1 -8277.337,E2 -8277.337} C_VEL
LIN {X 0,Y 453.824,Z 294.569,A -85,B 0,C 180,E1 -8280,E2 -8280} C_VEL
LIN {X 0,Y 453.732,Z 294.59,A -85,B 0,C 180,E1 -8282.663,E2 -8282.663} C_VEL
LIN {X 0,Y 453.653,Z 294.593,A -85,B 0,C 180,E1 -8286.226,E2 -8286.226} C_VEL
LIN {X 0,Y 453.587,Z 294.608,A -85,B 0,C 180,E1 -8288.913,E2 -8288.913} C_VEL
LIN {X 0,Y 453.564,Z 294.61,A -85,B 0,C 180,E1 -8292.529,E2 -8292.529} C_VEL
LIN {X 0,Y 453.544,Z 294.605,A -85,B 0,C 180,E1 -8296.196,E2 -8296.196} C_VEL
LIN {X 0,Y 453.517,Z 294.618,A -85,B 0,C 180,E1 -8299.039,E2 -8299.039} C_VEL
LIN {X 0,Y 453.476,Z 294.616,A -85,B 0,C 180,E1 -8301.836,E2 -8301.836} C_VEL
LIN {X 0,Y 453.489,Z 294.622,A -85,B 0,C 180,E1 -8304.736,E2 -8304.736} C_VEL
LIN {X 0,Y 453.489,Z 294.618,A -85,B 0,C 180,E1 -8307.949,E2 -8307.949} C_VEL
LIN {X 0,Y 453.475,Z 294.623,A -85,B 0,C 180,E1 -8310.76,E2 -8310.76} C_VEL
LIN {X 0,Y 453.476,Z 294.624,A -85,B 0,C 180,E1 -8313.913,E2 -8313.913} C_VEL
LIN {X 0,Y 453.448,Z 294.628,A -85,B 0,C 180,E1 -8317.19,E2 -8317.19} C_VEL
LIN {X 0,Y 453.493,Z 294.621,A -85,B 0,C 180,E1 -8320.609,E2 -8320.609} C_VEL
LIN {X 0,Y 453.454,Z 294.623,A -85,B 0,C 180,E1 -8323.244,E2 -8323.244} C_VEL
LIN {X 0,Y 453.453,Z 294.62,A -85,B 0,C 180,E1 -8326.305,E2 -8326.305} C_VEL
LIN {X 0,Y 453.47,Z 294.72,A -85,B 0,C 180,E1 -8326.622,E2 -8326.622} C_VEL
LIN {X 0,Y 456.434,Z 306.407,A -85,B 0,C 180,E1 -8329.894,E2 -8329.894} C_VEL
LIN {X 0,Y 459.487,Z 318.621,A -85,B 0,C 180,E1 -8333.077,E2 -8333.077} C_VEL
LIN {X 0,Y 460.483,Z 322.988,A -85,B 0,C 180,E1 -8334.163,E2 -8334.163} C_VEL
LIN {X 0,Y 458.925,Z 337.922,A -85,B 0,C 180,E1 -8337.381,E2 -8337.381} C_VEL
LIN {X 0,Y 457.486,Z 353.211,A -85,B 0,C 180,E1 -8340.555,E2 -8340.555} C_VEL
LIN {X 0,Y 456.367,Z 367.641,A -85,B 0,C 180,E1 -8343.475,E2 -8343.475} C_VEL
LIN {X 0,Y 455.236,Z 384.617,A -85,B 0,C 180,E1 -8346.817,E2 -8346.817} C_VEL
LIN {X 0,Y 454.984,Z 389.711,A -85,B 0,C 180,E1 -8347.807,E2 -8347.807} C_VEL
LIN {X 0,Y 457.888,Z 407.564,A -85,B 0,C 180,E1 -8348.3,E2 -8348.3} C_VEL
LIN {X 0,Y 459.505,Z 420.617,A -85,B 0,C 180,E1 -8348.762,E2 -8348.762} C_VEL
LIN {X 0,Y 458.854,Z 434.34,A -85,B 0,C 180,E1 -8349.299,E2 -8349.299} C_VEL
LIN {X 0,Y 458.041,Z 448.746,A -85,B 0,C 180,E1 -8350.038,E2 -8350.038} C_VEL
LIN {X 0,Y 457.123,Z 462.495,A -85,B 0,C 180,E1 -8350.931,E2 -8350.931} C_VEL
LIN {X 0,Y 456.264,Z 475.144,A -85,B 0,C 180,E1 -8351.941,E2 -8351.941} C_VEL
LIN {X 0,Y 455.491,Z 486.84,A -85,B 0,C 180,E1 -8353.063,E2 -8353.063} C_VEL
LIN {X 0,Y 454.714,Z 497.797,A -85,B 0,C 180,E1 -8354.307,E2 -8354.307} C_VEL
LIN {X 0,Y 454.061,Z 507.892,A -85,B 0,C 180,E1 -8355.662,E2 -8355.662} C_VEL
LIN {X 0,Y 453.488,Z 517.764,A -85,B 0,C 180,E1 -8357.242,E2 -8357.242} C_VEL
LIN {X 0,Y 453.175,Z 525.997,A -85,B 0,C 180,E1 -8358.822,E2 -8358.822} C_VEL
LIN {X 0,Y 452.856,Z 533.669,A -85,B 0,C 180,E1 -8360.622,E2 -8360.622} C_VEL
LIN {X 0,Y 452.746,Z 539.769,A -85,B 0,C 180,E1 -8362.418,E2 -8362.418} C_VEL
LIN {X 0,Y 452.76,Z 543.377,A -85,B 0,C 180,E1 -8363.762,E2 -8363.762} C_VEL
LIN {X 0,Y 452.711,Z 547.036,A -85,B 0,C 180,E1 -8365.548,E2 -8365.548} C_VEL
LIN {X 0,Y 452.766,Z 549.452,A -85,B 0,C 180,E1 -8367.331,E2 -8367.331} C_VEL
LIN {X 0,Y 452.68,Z 550.659,A -85,B 0,C 180,E1 -8369.111,E2 -8369.111} C_VEL
LIN {X 0,Y 452.679,Z 550.659,A -85,B 0,C 180,E1 -8370.89,E2 -8370.89} C_VEL
LIN {X 0,Y 452.771,Z 549.457,A -85,B 0,C 180,E1 -8372.669,E2 -8372.669} C_VEL
LIN {X 0,Y 452.795,Z 547.047,A -85,B 0,C 180,E1 -8374.451,E2 -8374.451} C_VEL
LIN {X 0,Y 452.779,Z 543.376,A -85,B 0,C 180,E1 -8376.238,E2 -8376.238} C_VEL
LIN {X 0,Y 452.807,Z 538.368,A -85,B 0,C 180,E1 -8378.03,E2 -8378.03} C_VEL
LIN {X 0,Y 452.923,Z 531.898,A -85,B 0,C 180,E1 -8379.828,E2 -8379.828} C_VEL
LIN {X 0,Y 453.212,Z 524.924,A -85,B 0,C 180,E1 -8381.404,E2 -8381.404} C_VEL
LIN {X 0,Y 453.581,Z 516.496,A -85,B 0,C 180,E1 -8382.984,E2 -8382.984} C_VEL
LIN {X 0,Y 454.163,Z 506.354,A -85,B 0,C 180,E1 -8384.564,E2 -8384.564} C_VEL
LIN {X 0,Y 454.855,Z 495.979,A -85,B 0,C 180,E1 -8385.918,E2 -8385.918} C_VEL
LIN {X 0,Y 455.742,Z 483.613,A -85,B 0,C 180,E1 -8387.269,E2 -8387.269} C_VEL
LIN {X 0,Y 456.555,Z 471.207,A -85,B 0,C 180,E1 -8388.395,E2 -8388.395} C_VEL
LIN {X 0,Y 457.461,Z 457.696,A -85,B 0,C 180,E1 -8389.404,E2 -8389.404} C_VEL
LIN {X 0,Y 458.424,Z 442.699,A -85,B 0,C 180,E1 -8390.296,E2 -8390.296} C_VEL
LIN {X 0,Y 459.172,Z 427.475,A -85,B 0,C 180,E1 -8390.989,E2 -8390.989} C_VEL
LIN {X 0,Y 459.383,Z 418.398,A -85,B 0,C 180,E1 -8391.313,E2 -8391.313} C_VEL
LIN {X 0,Y 457.768,Z 405.444,A -85,B 0,C 180,E1 -8391.759,E2 -8391.759} C_VEL
LIN {X 0,Y 455.102,Z 388.757,A -85,B 0,C 180,E1 -8392.195,E2 -8392.195} C_VEL
LIN {X 0,Y 454.752,Z 386.228,A -85,B 0,C 180,E1 -8392.286,E2 -8392.286} C_VEL
LIN {X 0,Y 455.586,Z 369.261,A -85,B 0,C 180,E1 -8395.591,E2 -8395.591} C_VEL
LIN {X 0,Y 456.629,Z 355.302,A -85,B 0,C 180,E1 -8398.498,E2 -8398.498} C_VEL
LIN {X 0,Y 458.107,Z 342.289,A -85,B 0,C 180,E1 -8401.44,E2 -8401.44} C_VEL
LIN {X 0,Y 460.053,Z 330.485,A -85,B 0,C 180,E1 -8404.419,E2 -8404.419} C_VEL
LIN {X 0,Y 461.015,Z 325.715,A -85,B 0,C 180,E1 -8405.754,E2 -8405.754} C_VEL
LIN {X 0,Y 460.814,Z 323.503,A -85,B 0,C 180,E1 -8406.499,E2 -8406.499} C_VEL
LIN {X 0,Y 459.307,Z 317.666,A -85,B 0,C 180,E1 -8408.856,E2 -8408.856} C_VEL
LIN {X 0,Y 458.057,Z 312.958,A -85,B 0,C 180,E1 -8411.281,E2 -8411.281} C_VEL
LIN {X 0,Y 457.079,Z 309.477,A -85,B 0,C 180,E1 -8413.782,E2 -8413.782} C_VEL
LIN {X 0,Y 456.381,Z 307.219,A -85,B 0,C 180,E1 -8416.367,E2 -8416.367} C_VEL
LIN {X 0,Y 455.95,Z 306.076,A -85,B 0,C 180,E1 -8419.051,E2 -8419.051} C_VEL
LIN {X 0,Y 455.676,Z 305.941,A -85,B 0,C 180,E1 -8421.908,E2 -8421.908} C_VEL
LIN {X 0,Y 455.482,Z 306.381,A -85,B 0,C 180,E1 -8424.103,E2 -8424.103} C_VEL
LIN {X 0,Y 455.182,Z 307.282,A -85,B 0,C 180,E1 -8426.487,E2 -8426.487} C_VEL
LIN {X 0,Y 454.802,Z 309.058,A -85,B 0,C 180,E1 -8429.925,E2 -8429.925} C_VEL
LIN {X 0,Y 454.521,Z 311.155,A -85,B 0,C 180,E1 -8433.358,E2 -8433.358} C_VEL
LIN {X 0,Y 454.35,Z 313.125,A -85,B 0,C 180,E1 -8436.286,E2 -8436.286} C_VEL
LIN {X 0,Y 454.187,Z 315.229,A -85,B 0,C 180,E1 -8439.152,E2 -8439.152} C_VEL
LIN {X 0,Y 454.013,Z 317.391,A -85,B 0,C 180,E1 -8441.965,E2 -8441.965} C_VEL
LIN {X 0,Y 453.975,Z 318.544,A -85,B 0,C 180,E1 -8443.396,E2 -8443.396} C_VEL
LIN {X 0,Y 458.852,Z 331.838,A -85,B 0,C 180,E1 -8444.225,E2 -8444.225} C_VEL
LIN {X 0,Y 458.329,Z 344.514,A -85,B 0,C 180,E1 -8444.89,E2 -8444.89} C_VEL
LIN {X 0,Y 457.773,Z 355.654,A -85,B 0,C 180,E1 -8445.636,E2 -8445.636} C_VEL
LIN {X 0,Y 457.082,Z 366.682,A -85,B 0,C 180,E1 -8446.552,E2 -8446.552} C_VEL
LIN {X 0,Y 456.457,Z 376.469,A -85,B 0,C 180,E1 -8447.552,E2 -8447.552} C_VEL
LIN {X 0,Y 455.808,Z 387.112,A -85,B 0,C 180,E1 -8448.888,E2 -8448.888} C_VEL
LIN {X 0,Y 455.111,Z 395.656,A -85,B 0,C 180,E1 -8450.22,E2 -8450.22} C_VEL
LIN {X 0,Y 454.643,Z 402.873,A -85,B 0,C 180,E1 -8451.625,E2 -8451.625} C_VEL
LIN {X 0,Y 454.29,Z 408.088,A -85,B 0,C 180,E1 -8452.891,E2 -8452.891} C_VEL
LIN {X 0,Y 453.958,Z 412.452,A -85,B 0,C 180,E1 -8454.225,E2 -8454.225} C_VEL
LIN {X 0,Y 453.656,Z 415.754,A -85,B 0,C 180,E1 -8455.558,E2 -8455.558} C_VEL
LIN {X 0,Y 453.711,Z 417.392,A -85,B 0,C 180,E1 -8456.448,E2 -8456.448} C_VEL
LIN {X 0,Y 453.528,Z 418.632,A -85,B 0,C 180,E1 -8457.336,E2 -8457.336} C_VEL
LIN {X 0,Y 453.354,Z 419.897,A -85,B 0,C 180,E1 -8459.112,E2 -8459.112} C_VEL
LIN {X 0,Y 453.329,Z 419.948,A -85,B 0,C 180,E1 -8460,E2 -8460} C_VEL
LIN {X 0,Y 453.336,Z 419.577,A -85,B 0,C 180,E1 -8460.888,E2 -8460.888} C_VEL
LIN {X 0,Y 453.203,Z 417.659,A -85,B 0,C 180,E1 -8462.667,E2 -8462.667} C_VEL
LIN {X 0,Y 453.322,Z 415.122,A -85,B 0,C 180,E1 -8464.001,E2 -8464.001} C_VEL
LIN {X 0,Y 453.473,Z 411.605,A -85,B 0,C 180,E1 -8465.336,E2 -8465.336} C_VEL
LIN {X 0,Y 453.785,Z 406.508,A -85,B 0,C 180,E1 -8466.797,E2 -8466.797} C_VEL
LIN {X 0,Y 454.064,Z 400.17,A -85,B 0,C 180,E1 -8468.232,E2 -8468.232} C_VEL
LIN {X 0,Y 454.414,Z 392.741,A -85,B 0,C 180,E1 -8469.571,E2 -8469.571} C_VEL
LIN {X 0,Y 454.765,Z 383.592,A -85,B 0,C 180,E1 -8470.913,E2 -8470.913} C_VEL
LIN {X 0,Y 455.332,Z 374.26,A -85,B 0,C 180,E1 -8472.027,E2 -8472.027} C_VEL
LIN {X 0,Y 455.818,Z 364.059,A -85,B 0,C 180,E1 -8473.032,E2 -8473.032} C_VEL
LIN {X 0,Y 456.273,Z 352.242,A -85,B 0,C 180,E1 -8473.976,E2 -8473.976} C_VEL
LIN {X 0,Y 456.797,Z 339.759,A -85,B 0,C 180,E1 -8474.763,E2 -8474.763} C_VEL
LIN {X 0,Y 456.947,Z 326.972,A -85,B 0,C 180,E1 -8475.382,E2 -8475.382} C_VEL
LIN {X 0,Y 453.294,Z 313.287,A -85,B 0,C 180,E1 -8475.998,E2 -8475.998} C_VEL
LIN {X 0,Y 452.893,Z 311.504,A -85,B 0,C 180,E1 -8476.082,E2 -8476.082} C_VEL
LIN {X 0,Y 452.915,Z 308.242,A -85,B 0,C 180,E1 -8479.018,E2 -8479.018} C_VEL
LIN {X 0,Y 452.921,Z 305.159,A -85,B 0,C 180,E1 -8481.864,E2 -8481.864} C_VEL
LIN {X 0,Y 452.941,Z 302.01,A -85,B 0,C 180,E1 -8484.768,E2 -8484.768} C_VEL
LIN {X 0,Y 452.963,Z 298.766,A -85,B 0,C 180,E1 -8487.823,E2 -8487.823} C_VEL
LIN {X 0,Y 452.959,Z 295.603,A -85,B 0,C 180,E1 -8490.799,E2 -8490.799} C_VEL
LIN {X 0,Y 452.989,Z 294.688,A -85,B 0,C 180,E1 -8491.837,E2 -8491.837} C_VEL
LIN {X 0,Y 453.364,Z 294.639,A -85,B 0,C 180,E1 -8495,E2 -8495} C_VEL
LIN {X 0,Y 453.466,Z 294.623,A -85,B 0,C 180,E1 -8498.312,E2 -8498.312} C_VEL
LIN {X 0,Y 453.497,Z 294.62,A -85,B 0,C 180,E1 -8500.609,E2 -8500.609} C_VEL
LIN {X 0,Y 453.455,Z 294.621,A -85,B 0,C 180,E1 -8503.244,E2 -8503.244} C_VEL
LIN {X 0,Y 453.46,Z 294.625,A -85,B 0,C 180,E1 -8505.778,E2 -8505.778} C_VEL
LIN {X 0,Y 453.441,Z 294.735,A -85,B 0,C 180,E1 -8508.945,E2 -8508.945} C_VEL
LIN {X 0,Y 453.499,Z 298.656,A -85,B 0,C 180,E1 -8511.691,E2 -8511.691} C_VEL
LIN {X 0,Y 453.442,Z 303.246,A -85,B 0,C 180,E1 -8515.007,E2 -8515.007} C_VEL
LIN {X 0,Y 453.352,Z 307.54,A -85,B 0,C 180,E1 -8518.191,E2 -8518.191} C_VEL
LIN {X 0,Y 453.296,Z 311.754,A -85,B 0,C 180,E1 -8521.273,E2 -8521.273} C_VEL
LIN {X 0,Y 453.26,Z 316.036,A -85,B 0,C 180,E1 -8524.268,E2 -8524.268} C_VEL
LIN {X 0,Y 453.245,Z 321.168,A -85,B 0,C 180,E1 -8527.566,E2 -8527.566} C_VEL
LIN {X 0,Y 459.469,Z 339.208,A -85,B 0,C 180,E1 -8528.334,E2 -8528.334} C_VEL
LIN {X 0,Y 460.923,Z 344.397,A -85,B 0,C 180,E1 -8528.583,E2 -8528.583} C_VEL
LIN {X 0,Y 460.397,Z 359.268,A -85,B 0,C 180,E1 -8529.173,E2 -8529.173} C_VEL
LIN {X 0,Y 459.711,Z 372.831,A -85,B 0,C 180,E1 -8529.88,E2 -8529.88} C_VEL
LIN {X 0,Y 458.938,Z 386.428,A -85,B 0,C 180,E1 -8530.777,E2 -8530.777} C_VEL
LIN {X 0,Y 458.005,Z 398.897,A -85,B 0,C 180,E1 -8531.781,E2 -8531.781} C_VEL
LIN {X 0,Y 457.899,Z 401.081,A -85,B 0,C 180,E1 -8531.979,E2 -8531.979} C_VEL
LIN {X 0,Y 456.961,Z 405.852,A -85,B 0,C 180,E1 -8532.4,E2 -8532.4} C_VEL
LIN {X 0,Y 453.594,Z 413.506,A -85,B 0,C 180,E1 -8533.073,E2 -8533.073} C_VEL
LIN {X 0,Y 450.196,Z 420.849,A -85,B 0,C 180,E1 -8533.802,E2 -8533.802} C_VEL
LIN {X 0,Y 449.187,Z 425.018,A -85,B 0,C 180,E1 -8534.319,E2 -8534.319} C_VEL
LIN {X 0,Y 448.329,Z 434.478,A -85,B 0,C 180,E1 -8535.706,E2 -8535.706} C_VEL
LIN {X 0,Y 447.632,Z 443.577,A -85,B 0,C 180,E1 -8537.302,E2 -8537.302} C_VEL
LIN {X 0,Y 447.055,Z 450.171,A -85,B 0,C 180,E1 -8538.667,E2 -8538.667} C_VEL
LIN {X 0,Y 446.495,Z 457.407,A -85,B 0,C 180,E1 -8540.487,E2 -8540.487} C_VEL
LIN {X 0,Y 446.119,Z 463.138,A -85,B 0,C 180,E1 -8542.304,E2 -8542.304} C_VEL
LIN {X 0,Y 445.899,Z 466.523,A -85,B 0,C 180,E1 -8543.665,E2 -8543.665} C_VEL
LIN {X 0,Y 445.758,Z 469.967,A -85,B 0,C 180,E1 -8545.478,E2 -8545.478} C_VEL
LIN {X 0,Y 445.673,Z 472.24,A -85,B 0,C 180,E1 -8547.288,E2 -8547.288} C_VEL
LIN {X 0,Y 445.456,Z 473.412,A -85,B 0,C 180,E1 -8549.096,E2 -8549.096} C_VEL
LIN {X 0,Y 445.456,Z 473.427,A -85,B 0,C 180,E1 -8550.904,E2 -8550.904} C_VEL
LIN {X 0,Y 445.673,Z 472.314,A -85,B 0,C 180,E1 -8552.711,E2 -8552.711} C_VEL
LIN {X 0,Y 445.757,Z 470.104,A -85,B 0,C 180,E1 -8554.521,E2 -8554.521} C_VEL
LIN {X 0,Y 445.895,Z 466.732,A -85,B 0,C 180,E1 -8556.334,E2 -8556.334} C_VEL
LIN {X 0,Y 446.201,Z 462.098,A -85,B 0,C 180,E1 -8558.149,E2 -8558.149} C_VEL
LIN {X 0,Y 446.583,Z 456.084,A -85,B 0,C 180,E1 -8559.968,E2 -8559.968} C_VEL
LIN {X 0,Y 447.207,Z 448.503,A -85,B 0,C 180,E1 -8561.788,E2 -8561.788} C_VEL
LIN {X 0,Y 447.764,Z 440.853,A -85,B 0,C 180,E1 -8563.31,E2 -8563.31} C_VEL
LIN {X 0,Y 448.572,Z 432.175,A -85,B 0,C 180,E1 -8564.75,E2 -8564.75} C_VEL
LIN {X 0,Y 449.45,Z 422.423,A -85,B 0,C 180,E1 -8566.114,E2 -8566.114} C_VEL
LIN {X 0,Y 450.418,Z 410.506,A -85,B 0,C 180,E1 -8567.516,E2 -8567.516} C_VEL
LIN {X 0,Y 451.46,Z 397.989,A -85,B 0,C 180,E1 -8568.728,E2 -8568.728} C_VEL
LIN {X 0,Y 452.36,Z 385.172,A -85,B 0,C 180,E1 -8569.75,E2 -8569.75} C_VEL
LIN {X 0,Y 453.267,Z 371.096,A -85,B 0,C 180,E1 -8570.655,E2 -8570.655} C_VEL
LIN {X 0,Y 453.919,Z 356.901,A -85,B 0,C 180,E1 -8571.373,E2 -8571.373} C_VEL
LIN {X 0,Y 454.237,Z 345.453,A -85,B 0,C 180,E1 -8571.825,E2 -8571.825} C_VEL
LIN {X 0,Y 450.112,Z 332.612,A -85,B 0,C 180,E1 -8572.441,E2 -8572.441} C_VEL
LIN {X 0,Y 446.228,Z 321.762,A -85,B 0,C 180,E1 -8572.882,E2 -8572.882} C_VEL
LIN {X 0,Y 446.242,Z 316.662,A -85,B 0,C 180,E1 -8576.166,E2 -8576.166} C_VEL
LIN {X 0,Y 446.285,Z 312.269,A -85,B 0,C 180,E1 -8579.221,E2 -8579.221} C_VEL
LIN {X 0,Y 446.328,Z 307.987,A -85,B 0,C 180,E1 -8582.369,E2 -8582.369} C_VEL
LIN {X 0,Y 446.407,Z 304.385,A -85,B 0,C 180,E1 -8585.049,E2 -8585.049} C_VEL
LIN {X 0,Y 446.473,Z 300.219,A -85,B 0,C 180,E1 -8588.088,E2 -8588.088} C_VEL
LIN {X 0,Y 446.442,Z 296.206,A -85,B 0,C 180,E1 -8590.92,E2 -8590.92} C_VEL
LIN {X 0,Y 446.392,Z 295.513,A -85,B 0,C 180,E1 -8591.545,E2 -8591.545} C_VEL
LIN {X 0,Y 446.453,Z 295.502,A -85,B 0,C 180,E1 -8595.103,E2 -8595.103} C_VEL
LIN {X 0,Y 446.428,Z 295.501,A -85,B 0,C 180,E1 -8598.609,E2 -8598.609} C_VEL
LIN {X 0,Y 446.412,Z 295.506,A -85,B 0,C 180,E1 -8601.921,E2 -8601.921} C_VEL
LIN {X 0,Y 446.43,Z 295.501,A -85,B 0,C 180,E1 -8605.477,E2 -8605.477} C_VEL
LIN {X 0,Y 446.415,Z 295.503,A -85,B 0,C 180,E1 -8608.699,E2 -8608.699} C_VEL
LIN {X 0,Y 446.423,Z 295.504,A -85,B 0,C 180,E1 -8611.836,E2 -8611.836} C_VEL
LIN {X 0,Y 446.433,Z 295.496,A -85,B 0,C 180,E1 -8614.846,E2 -8614.846} C_VEL
LIN {X 0,Y 446.449,Z 295.491,A -85,B 0,C 180,E1 -8618.245,E2 -8618.245} C_VEL
LIN {X 0,Y 446.449,Z 295.5,A -85,B 0,C 180,E1 -8621.649,E2 -8621.649} C_VEL
LIN {X 0,Y 446.509,Z 295.487,A -85,B 0,C 180,E1 -8624.48,E2 -8624.48} C_VEL
LIN {X 0,Y 446.518,Z 295.481,A -85,B 0,C 180,E1 -8628.193,E2 -8628.193} C_VEL
LIN {X 0,Y 446.531,Z 295.487,A -85,B 0,C 180,E1 -8630.944,E2 -8630.944} C_VEL
LIN {X 0,Y 446.611,Z 295.468,A -85,B 0,C 180,E1 -8633.676,E2 -8633.676} C_VEL
LIN {X 0,Y 446.689,Z 295.468,A -85,B 0,C 180,E1 -8637.294,E2 -8637.294} C_VEL
LIN {X 0,Y 446.793,Z 295.444,A -85,B 0,C 180,E1 -8640,E2 -8640} C_VEL
LIN {X 0,Y 446.679,Z 295.468,A -85,B 0,C 180,E1 -8642.705,E2 -8642.705} C_VEL
LIN {X 0,Y 446.623,Z 295.469,A -85,B 0,C 180,E1 -8646.324,E2 -8646.324} C_VEL
LIN {X 0,Y 446.534,Z 295.485,A -85,B 0,C 180,E1 -8649.055,E2 -8649.055} C_VEL
LIN {X 0,Y 446.521,Z 295.487,A -85,B 0,C 180,E1 -8652.73,E2 -8652.73} C_VEL
LIN {X 0,Y 446.488,Z 295.483,A -85,B 0,C 180,E1 -8656.459,E2 -8656.459} C_VEL
LIN {X 0,Y 446.468,Z 295.495,A -85,B 0,C 180,E1 -8659.303,E2 -8659.303} C_VEL
LIN {X 0,Y 446.417,Z 295.496,A -85,B 0,C 180,E1 -8662.2,E2 -8662.2} C_VEL
LIN {X 0,Y 446.431,Z 295.5,A -85,B 0,C 180,E1 -8665.154,E2 -8665.154} C_VEL
LIN {X 0,Y 446.439,Z 295.498,A -85,B 0,C 180,E1 -8668.182,E2 -8668.182} C_VEL
LIN {X 0,Y 446.415,Z 295.502,A -85,B 0,C 180,E1 -8671.3,E2 -8671.3} C_VEL
LIN {X 0,Y 446.427,Z 295.5,A -85,B 0,C 180,E1 -8674.523,E2 -8674.523} C_VEL
LIN {X 0,Y 446.41,Z 295.504,A -85,B 0,C 180,E1 -8678.078,E2 -8678.078} C_VEL
LIN {X 0,Y 446.426,Z 295.5,A -85,B 0,C 180,E1 -8680.918,E2 -8680.918} C_VEL
LIN {X 0,Y 446.399,Z 295.5,A -85,B 0,C 180,E1 -8683.846,E2 -8683.846} C_VEL
LIN {X 0,Y 446.429,Z 295.619,A -85,B 0,C 180,E1 -8686.123,E2 -8686.123} C_VEL
LIN {X 0,Y 449.264,Z 306.895,A -85,B 0,C 180,E1 -8689.349,E2 -8689.349} C_VEL
LIN {X 0,Y 452.165,Z 318.413,A -85,B 0,C 180,E1 -8692.438,E2 -8692.438} C_VEL
LIN {X 0,Y 453.579,Z 324.265,A -85,B 0,C 180,E1 -8693.929,E2 -8693.929} C_VEL
LIN {X 0,Y 453.017,Z 330.419,A -85,B 0,C 180,E1 -8695.308,E2 -8695.308} C_VEL
LIN {X 0,Y 451.622,Z 343.069,A -85,B 0,C 180,E1 -8698.056,E2 -8698.056} C_VEL
LIN {X 0,Y 450.181,Z 358.559,A -85,B 0,C 180,E1 -8701.311,E2 -8701.311} C_VEL
LIN {X 0,Y 448.962,Z 374.167,A -85,B 0,C 180,E1 -8704.502,E2 -8704.502} C_VEL
LIN {X 0,Y 448.02,Z 388.894,A -85,B 0,C 180,E1 -8707.444,E2 -8707.444} C_VEL
LIN {X 0,Y 451.012,Z 406.687,A -85,B 0,C 180,E1 -8707.943,E2 -8707.943} C_VEL
LIN {X 0,Y 452.796,Z 421.481,A -85,B 0,C 180,E1 -8708.487,E2 -8708.487} C_VEL
LIN {X 0,Y 452.025,Z 436.498,A -85,B 0,C 180,E1 -8709.107,E2 -8709.107} C_VEL
LIN {X 0,Y 451.191,Z 450.079,A -85,B 0,C 180,E1 -8709.841,E2 -8709.841} C_VEL
LIN {X 0,Y 450.232,Z 463.473,A -85,B 0,C 180,E1 -8710.746,E2 -8710.746} C_VEL
LIN {X 0,Y 449.254,Z 477.103,A -85,B 0,C 180,E1 -8711.886,E2 -8711.886} C_VEL
LIN {X 0,Y 448.411,Z 488.891,A -85,B 0,C 180,E1 -8713.077,E2 -8713.077} C_VEL
LIN {X 0,Y 447.524,Z 500.782,A -85,B 0,C 180,E1 -8714.516,E2 -8714.516} C_VEL
LIN {X 0,Y 446.804,Z 511.752,A -85,B 0,C 180,E1 -8716.121,E2 -8716.121} C_VEL
LIN {X 0,Y 446.216,Z 520.731,A -85,B 0,C 180,E1 -8717.695,E2 -8717.695} C_VEL
LIN {X 0,Y 446.075,Z 527.449,A -85,B 0,C 180,E1 -8719.102,E2 -8719.102} C_VEL
LIN {X 0,Y 445.742,Z 534.711,A -85,B 0,C 180,E1 -8720.929,E2 -8720.929} C_VEL
LIN {X 0,Y 445.673,Z 540.436,A -85,B 0,C 180,E1 -8722.753,E2 -8722.753} C_VEL
LIN {X 0,Y 445.669,Z 544.758,A -85,B 0,C 180,E1 -8724.571,E2 -8724.571} C_VEL
LIN {X 0,Y 445.687,Z 547.789,A -85,B 0,C 180,E1 -8726.384,E2 -8726.384} C_VEL
LIN {X 0,Y 445.659,Z 549.596,A -85,B 0,C 180,E1 -8728.193,E2 -8728.193} C_VEL
LIN {X 0,Y 445.606,Z 550.208,A -85,B 0,C 180,E1 -8730,E2 -8730} C_VEL
LIN {X 0,Y 445.649,Z 549.597,A -85,B 0,C 180,E1 -8731.808,E2 -8731.808} C_VEL
LIN {X 0,Y 445.709,Z 547.796,A -85,B 0,C 180,E1 -8733.616,E2 -8733.616} C_VEL
LIN {X 0,Y 445.711,Z 544.763,A -85,B 0,C 180,E1 -8735.429,E2 -8735.429} C_VEL
LIN {X 0,Y 445.684,Z 540.431,A -85,B 0,C 180,E1 -8737.248,E2 -8737.248} C_VEL
LIN {X 0,Y 445.755,Z 534.71,A -85,B 0,C 180,E1 -8739.072,E2 -8739.072} C_VEL
LIN {X 0,Y 446.09,Z 527.453,A -85,B 0,C 180,E1 -8740.898,E2 -8740.898} C_VEL
LIN {X 0,Y 446.355,Z 519.554,A -85,B 0,C 180,E1 -8742.523,E2 -8742.523} C_VEL
LIN {X 0,Y 446.9,Z 510.296,A -85,B 0,C 180,E1 -8744.108,E2 -8744.108} C_VEL
LIN {X 0,Y 447.522,Z 500.772,A -85,B 0,C 180,E1 -8745.484,E2 -8745.484} C_VEL
LIN {X 0,Y 448.454,Z 488.698,A -85,B 0,C 180,E1 -8746.942,E2 -8746.942} C_VEL
LIN {X 0,Y 449.356,Z 475.816,A -85,B 0,C 180,E1 -8748.229,E2 -8748.229} C_VEL
LIN {X 0,Y 450.294,Z 463.454,A -85,B 0,C 180,E1 -8749.251,E2 -8749.251} C_VEL
LIN {X 0,Y 451.223,Z 450.055,A -85,B 0,C 180,E1 -8750.158,E2 -8750.158} C_VEL
LIN {X 0,Y 452.097,Z 435.307,A -85,B 0,C 180,E1 -8750.95,E2 -8750.95} C_VEL
LIN {X 0,Y 452.761,Z 419.792,A -85,B 0,C 180,E1 -8751.576,E2 -8751.576} C_VEL
LIN {X 0,Y 451.258,Z 407.503,A -85,B 0,C 180,E1 -8752.021,E2 -8752.021} C_VEL
LIN {X 0,Y 449.132,Z 393.198,A -85,B 0,C 180,E1 -8752.424,E2 -8752.424} C_VEL
LIN {X 0,Y 447.782,Z 385.514,A -85,B 0,C 180,E1 -8752.637,E2 -8752.637} C_VEL
LIN {X 0,Y 448.701,Z 368.69,A -85,B 0,C 180,E1 -8756.013,E2 -8756.013} C_VEL
LIN {X 0,Y 450.02,Z 353.976,A -85,B 0,C 180,E1 -8759.186,E2 -8759.186} C_VEL
LIN {X 0,Y 451.451,Z 342.232,A -85,B 0,C 180,E1 -8761.958,E2 -8761.958} C_VEL
LIN {X 0,Y 453.609,Z 330.742,A -85,B 0,C 180,E1 -8764.978,E2 -8764.978} C_VEL
LIN {X 0,Y 454.281,Z 327.25,A -85,B 0,C 180,E1 -8766.007,E2 -8766.007} C_VEL
LIN {X 0,Y 453.296,Z 322.62,A -85,B 0,C 180,E1 -8767.748,E2 -8767.748} C_VEL
LIN {X 0,Y 451.845,Z 317.06,A -85,B 0,C 180,E1 -8770.346,E2 -8770.346} C_VEL
LIN {X 0,Y 450.708,Z 313.041,A -85,B 0,C 180,E1 -8772.872,E2 -8772.872} C_VEL
LIN {X 0,Y 449.928,Z 310.345,A -85,B 0,C 180,E1 -8775.339,E2 -8775.339} C_VEL
LIN {X 0,Y 449.42,Z 308.762,A -85,B 0,C 180,E1 -8777.745,E2 -8777.745} C_VEL
LIN {X 0,Y 449.092,Z 308.071,A -85,B 0,C 180,E1 -8780.087,E2 -8780.087} C_VEL
LIN {X 0,Y 448.797,Z 308.091,A -85,B 0,C 180,E1 -8783.001,E2 -8783.001} C_VEL
LIN {X 0,Y 448.452,Z 308.798,A -85,B 0,C 180,E1 -8785.655,E2 -8785.655} C_VEL
LIN {X 0,Y 448.005,Z 310.193,A -85,B 0,C 180,E1 -8788.823,E2 -8788.823} C_VEL
LIN {X 0,Y 447.714,Z 311.856,A -85,B 0,C 180,E1 -8791.906,E2 -8791.906} C_VEL
LIN {X 0,Y 447.504,Z 313.745,A -85,B 0,C 180,E1 -8794.911,E2 -8794.911} C_VEL
LIN {X 0,Y 447.314,Z 315.84,A -85,B 0,C 180,E1 -8797.97,E2 -8797.97} C_VEL
LIN {X 0,Y 447.164,Z 317.883,A -85,B 0,C 180,E1 -8800.728,E2 -8800.728} C_VEL
LIN {X 0,Y 447.065,Z 319.834,A -85,B 0,C 180,E1 -8803.018,E2 -8803.018} C_VEL
LIN {X 0,Y 451.855,Z 332.254,A -85,B 0,C 180,E1 -8803.831,E2 -8803.831} C_VEL
LIN {X 0,Y 452.272,Z 334.437,A -85,B 0,C 180,E1 -8803.967,E2 -8803.967} C_VEL
LIN {X 0,Y 451.7,Z 346.944,A -85,B 0,C 180,E1 -8804.663,E2 -8804.663} C_VEL
LIN {X 0,Y 451.015,Z 359.476,A -85,B 0,C 180,E1 -8805.563,E2 -8805.563} C_VEL
LIN {X 0,Y 450.251,Z 370.824,A -85,B 0,C 180,E1 -8806.574,E2 -8806.574} C_VEL
LIN {X 0,Y 449.562,Z 380.114,A -85,B 0,C 180,E1 -8807.587,E2 -8807.587} C_VEL
LIN {X 0,Y 448.846,Z 390.162,A -85,B 0,C 180,E1 -8808.942,E2 -8808.942} C_VEL
LIN {X 0,Y 448.251,Z 398.297,A -85,B 0,C 180,E1 -8810.297,E2 -8810.297} C_VEL
LIN {X 0,Y 447.774,Z 403.86,A -85,B 0,C 180,E1 -8811.423,E2 -8811.423} C_VEL
LIN {X 0,Y 447.362,Z 409.368,A -85,B 0,C 180,E1 -8812.78,E2 -8812.78} C_VEL
LIN {X 0,Y 447.009,Z 413.691,A -85,B 0,C 180,E1 -8814.135,E2 -8814.135} C_VEL
LIN {X 0,Y 446.706,Z 416.953,A -85,B 0,C 180,E1 -8815.488,E2 -8815.488} C_VEL
LIN {X 0,Y 446.726,Z 418.57,A -85,B 0,C 180,E1 -8816.392,E2 -8816.392} C_VEL
LIN {X 0,Y 446.54,Z 419.776,A -85,B 0,C 180,E1 -8817.294,E2 -8817.294} C_VEL
LIN {X 0,Y 446.34,Z 420.99,A -85,B 0,C 180,E1 -8819.098,E2 -8819.098} C_VEL
LIN {X 0,Y 446.312,Z 421.011,A -85,B 0,C 180,E1 -8820,E2 -8820} C_VEL
LIN {X 0,Y 446.319,Z 420.605,A -85,B 0,C 180,E1 -8820.902,E2 -8820.902} C_VEL
LIN {X 0,Y 446.179,Z 418.637,A -85,B 0,C 180,E1 -8822.709,E2 -8822.709} C_VEL
LIN {X 0,Y 446.308,Z 416.053,A -85,B 0,C 180,E1 -8824.064,E2 -8824.064} C_VEL
LIN {X 0,Y 446.474,Z 412.488,A -85,B 0,C 180,E1 -8825.42,E2 -8825.42} C_VEL
LIN {X 0,Y 446.775,Z 407.645,A -85,B 0,C 180,E1 -8826.827,E2 -8826.827} C_VEL
LIN {X 0,Y 447.097,Z 400.948,A -85,B 0,C 180,E1 -8828.361,E2 -8828.361} C_VEL
LIN {X 0,Y 447.452,Z 393.462,A -85,B 0,C 180,E1 -8829.721,E2 -8829.721} C_VEL
LIN {X 0,Y 447.829,Z 384.248,A -85,B 0,C 180,E1 -8831.084,E2 -8831.084} C_VEL
LIN {X 0,Y 448.413,Z 374.865,A -85,B 0,C 180,E1 -8832.215,E2 -8832.215} C_VEL
LIN {X 0,Y 448.951,Z 363.303,A -85,B 0,C 180,E1 -8833.35,E2 -8833.35} C_VEL
LIN {X 0,Y 449.495,Z 350.964,A -85,B 0,C 180,E1 -8834.321,E2 -8834.321} C_VEL
LIN {X 0,Y 449.975,Z 338.055,A -85,B 0,C 180,E1 -8835.108,E2 -8835.108} C_VEL
LIN {X 0,Y 450.178,Z 328.666,A -85,B 0,C 180,E1 -8835.565,E2 -8835.565} C_VEL
LIN {X 0,Y 446.484,Z 314.596,A -85,B 0,C 180,E1 -8836.221,E2 -8836.221} C_VEL
LIN {X 0,Y 445.83,Z 312.026,A -85,B 0,C 180,E1 -8836.339,E2 -8836.339} C_VEL
LIN {X 0,Y 445.87,Z 308.707,A -85,B 0,C 180,E1 -8839.33,E2 -8839.33} C_VEL
LIN {X 0,Y 445.863,Z 305.555,A -85,B 0,C 180,E1 -8842.229,E2 -8842.229} C_VEL
LIN {X 0,Y 445.872,Z 302.361,A -85,B 0,C 180,E1 -8845.188,E2 -8845.188} C_VEL
LIN {X 0,Y 445.912,Z 299.141,A -85,B 0,C 180,E1 -8848.218,E2 -8848.218} C_VEL
LIN {X 0,Y 445.942,Z 295.852,A -85,B 0,C 180,E1 -8851.337,E2 -8851.337} C_VEL
LIN {X 0,Y 446.031,Z 295.554,A -85,B 0,C 180,E1 -8852.394,E2 -8852.394} C_VEL
LIN {X 0,Y 446.342,Z 295.513,A -85,B 0,C 180,E1 -8855.633,E2 -8855.633} C_VEL
LIN {X 0,Y 446.458,Z 295.498,A -85,B 0,C 180,E1 -8859.026,E2 -8859.026} C_VEL
LIN {X 0,Y 446.437,Z 295.498,A -85,B 0,C 180,E1 -8862.277,E2 -8862.277} C_VEL
LIN {X 0,Y 446.452,Z 295.496,A -85,B 0,C 180,E1 -8865.104,E2 -8865.104} C_VEL
LIN {X 0,Y 446.408,Z 295.565,A -85,B 0,C 180,E1 -8868.743,E2 -8868.743} C_VEL
LIN {X 0,Y 446.479,Z 298.733,A -85,B 0,C 180,E1 -8870.976,E2 -8870.976} C_VEL
LIN {X 0,Y 446.404,Z 303.44,A -85,B 0,C 180,E1 -8874.372,E2 -8874.372} C_VEL
LIN {X 0,Y 446.33,Z 307.837,A -85,B 0,C 180,E1 -8877.631,E2 -8877.631} C_VEL
LIN {X 0,Y 446.284,Z 312.138,A -85,B 0,C 180,E1 -8880.779,E2 -8880.779} C_VEL
LIN {X 0,Y 446.226,Z 316.548,A -85,B 0,C 180,E1 -8883.863,E2 -8883.863} C_VEL
LIN {X 0,Y 446.238,Z 321.734,A -85,B 0,C 180,E1 -8887.2,E2 -8887.2} C_VEL
LIN {X 0,Y 452.371,Z 339.196,A -85,B 0,C 180,E1 -8887.959,E2 -8887.959} C_VEL
LIN {X 0,Y 454.338,Z 346.419,A -85,B 0,C 180,E1 -8888.308,E2 -8888.308} C_VEL
LIN {X 0,Y 453.778,Z 360.285,A -85,B 0,C 180,E1 -8888.876,E2 -8888.876} C_VEL
LIN {X 0,Y 453.093,Z 373.422,A -85,B 0,C 180,E1 -8889.574,E2 -8889.574} C_VEL
LIN {X 0,Y 452.28,Z 387.024,A -85,B 0,C 180,E1 -8890.483,E2 -8890.483} C_VEL
LIN {X 0,Y 451.308,Z 399.496,A -85,B 0,C 180,E1 -8891.501,E2 -8891.501} C_VEL
LIN {X 0,Y 450.266,Z 412.077,A -85,B 0,C 180,E1 -8892.749,E2 -8892.749} C_VEL
LIN {X 0,Y 449.312,Z 423.465,A -85,B 0,C 180,E1 -8894.113,E2 -8894.113} C_VEL
LIN {X 0,Y 449.187,Z 425.018,A -85,B 0,C 180,E1 -8894.319,E2 -8894.319} C_VEL
LIN {X 0,Y 448.22,Z 429.087,A -85,B 0,C 180,E1 -8894.851,E2 -8894.851} C_VEL
LIN {X 0,Y 444.901,Z 435.542,A -85,B 0,C 180,E1 -8895.717,E2 -8895.717} C_VEL
LIN {X 0,Y 441.588,Z 441.646,A -85,B 0,C 180,E1 -8896.639,E2 -8896.639} C_VEL
LIN {X 0,Y 440.645,Z 444.982,A -85,B 0,C 180,E1 -8897.254,E2 -8897.254} C_VEL
LIN {X 0,Y 439.945,Z 452.726,A -85,B 0,C 180,E1 -8898.948,E2 -8898.948} C_VEL
LIN {X 0,Y 439.414,Z 459.568,A -85,B 0,C 180,E1 -8900.796,E2 -8900.796} C_VEL
LIN {X 0,Y 439.003,Z 464.945,A -85,B 0,C 180,E1 -8902.642,E2 -8902.642} C_VEL
LIN {X 0,Y 438.708,Z 469.011,A -85,B 0,C 180,E1 -8904.484,E2 -8904.484} C_VEL
LIN {X 0,Y 438.708,Z 471.85,A -85,B 0,C 180,E1 -8906.326,E2 -8906.326} C_VEL
LIN {X 0,Y 438.477,Z 473.573,A -85,B 0,C 180,E1 -8908.163,E2 -8908.163} C_VEL
LIN {X 0,Y 438.37,Z 474.174,A -85,B 0,C 180,E1 -8910,E2 -8910} C_VEL
LIN {X 0,Y 438.476,Z 473.617,A -85,B 0,C 180,E1 -8911.837,E2 -8911.837} C_VEL
LIN {X 0,Y 438.694,Z 471.954,A -85,B 0,C 180,E1 -8913.674,E2 -8913.674} C_VEL
LIN {X 0,Y 438.705,Z 469.181,A -85,B 0,C 180,E1 -8915.516,E2 -8915.516} C_VEL
LIN {X 0,Y 439.057,Z 465.182,A -85,B 0,C 180,E1 -8917.357,E2 -8917.357} C_VEL
LIN {X 0,Y 439.395,Z 459.878,A -85,B 0,C 180,E1 -8919.204,E2 -8919.204} C_VEL
LIN {X 0,Y 439.935,Z 453.106,A -85,B 0,C 180,E1 -8921.052,E2 -8921.052} C_VEL
LIN {X 0,Y 440.579,Z 445.845,A -85,B 0,C 180,E1 -8922.67,E2 -8922.67} C_VEL
LIN {X 0,Y 441.327,Z 437.083,A -85,B 0,C 180,E1 -8924.29,E2 -8924.29} C_VEL
LIN {X 0,Y 442.337,Z 426.472,A -85,B 0,C 180,E1 -8925.907,E2 -8925.907} C_VEL
LIN {X 0,Y 443.317,Z 415.565,A -85,B 0,C 180,E1 -8927.292,E2 -8927.292} C_VEL
LIN {X 0,Y 444.355,Z 403.578,A -85,B 0,C 180,E1 -8928.56,E2 -8928.56} C_VEL
LIN {X 0,Y 445.393,Z 390.339,A -85,B 0,C 180,E1 -8929.711,E2 -8929.711} C_VEL
LIN {X 0,Y 446.349,Z 377.386,A -85,B 0,C 180,E1 -8930.628,E2 -8930.628} C_VEL
LIN {X 0,Y 447.094,Z 363.832,A -85,B 0,C 180,E1 -8931.401,E2 -8931.401} C_VEL
LIN {X 0,Y 447.721,Z 349.131,A -85,B 0,C 180,E1 -8932.044,E2 -8932.044} C_VEL
LIN {X 0,Y 447.5,Z 346.597,A -85,B 0,C 180,E1 -8932.15,E2 -8932.15} C_VEL
LIN {X 0,Y 443.108,Z 332.945,A -85,B 0,C 180,E1 -8932.82,E2 -8932.82} C_VEL
LIN {X 0,Y 439.248,Z 322.305,A -85,B 0,C 180,E1 -8933.279,E2 -8933.279} C_VEL
LIN {X 0,Y 439.252,Z 317.128,A -85,B 0,C 180,E1 -8936.615,E2 -8936.615} C_VEL
LIN {X 0,Y 439.266,Z 312.653,A -85,B 0,C 180,E1 -8939.734,E2 -8939.734} C_VEL
LIN {X 0,Y 439.328,Z 308.286,A -85,B 0,C 180,E1 -8942.95,E2 -8942.95} C_VEL
LIN {X 0,Y 439.377,Z 303.775,A -85,B 0,C 180,E1 -8946.287,E2 -8946.287} C_VEL
LIN {X 0,Y 439.467,Z 300.614,A -85,B 0,C 180,E1 -8948.586,E2 -8948.586} C_VEL
LIN {X 0,Y 439.373,Z 296.387,A -85,B 0,C 180,E1 -8951.594,E2 -8951.594} C_VEL
LIN {X 0,Y 439.401,Z 296.381,A -85,B 0,C 180,E1 -8955.271,E2 -8955.271} C_VEL
